LIN {X 0,Y 572.631,Z 334.16,A -85,B 0,C 180,E1 -2364.976,E2 -2364.976} C_VEL
LIN {X 0,Y 569.788,Z 334.515,A -85,B 0,C 180,E1 -2365.927,E2 -2365.927} C_VEL
LIN {X 0,Y 567.355,Z 334.817,A -85,B 0,C 180,E1 -2366.692,E2 -2366.692} C_VEL
LIN {X 0,Y 566.3,Z 334.946,A -85,B 0,C 180,E1 -2367.283,E2 -2367.283} C_VEL
LIN {X 0,Y 566.21,Z 334.956,A -85,B 0,C 180,E1 -2367.484,E2 -2367.484} C_VEL
LIN {X 0,Y 566.206,Z 334.958,A -85,B 0,C 180,E1 -2369.769,E2 -2369.769} C_VEL
LIN {X 0,Y 566.212,Z 334.959,A -85,B 0,C 180,E1 -2372.43,E2 -2372.43} C_VEL
LIN {X 0,Y 566.189,Z 334.96,A -85,B 0,C 180,E1 -2374.99,E2 -2374.99} C_VEL
LIN {X 0,Y 566.203,Z 334.958,A -85,B 0,C 180,E1 -2377.461,E2 -2377.461} C_VEL
LIN {X 0,Y 566.235,Z 334.956,A -85,B 0,C 180,E1 -2380.197,E2 -2380.197} C_VEL
LIN {X 0,Y 566.207,Z 334.957,A -85,B 0,C 180,E1 -2383.054,E2 -2383.054} C_VEL
LIN {X 0,Y 566.209,Z 334.958,A -85,B 0,C 180,E1 -2386.048,E2 -2386.048} C_VEL
LIN {X 0,Y 566.19,Z 334.959,A -85,B 0,C 180,E1 -2388.861,E2 -2388.861} C_VEL
LIN {X 0,Y 566.189,Z 334.961,A -85,B 0,C 180,E1 -2391.636,E2 -2391.636} C_VEL
LIN {X 0,Y 566.158,Z 334.963,A -85,B 0,C 180,E1 -2394.307,E2 -2394.307} C_VEL
LIN {X 0,Y 566.237,Z 334.955,A -85,B 0,C 180,E1 -2396.898,E2 -2396.898} C_VEL
LIN {X 0,Y 566.18,Z 334.963,A -85,B 0,C 180,E1 -2399.407,E2 -2399.407} C_VEL
LIN {X 0,Y 566.219,Z 334.956,A -85,B 0,C 180,E1 -2401.857,E2 -2401.857} C_VEL
LIN {X 0,Y 566.222,Z 334.955,A -85,B 0,C 180,E1 -2404.251,E2 -2404.251} C_VEL
LIN {X 0,Y 566.18,Z 334.961,A -85,B 0,C 180,E1 -2406.718,E2 -2406.718} C_VEL
LIN {X 0,Y 566.215,Z 334.957,A -85,B 0,C 180,E1 -2409.662,E2 -2409.662} C_VEL
LIN {X 0,Y 566.208,Z 334.959,A -85,B 0,C 180,E1 -2412.668,E2 -2412.668} C_VEL
LIN {X 0,Y 566.242,Z 334.952,A -85,B 0,C 180,E1 -2415.626,E2 -2415.626} C_VEL
LIN {X 0,Y 566.243,Z 334.954,A -85,B 0,C 180,E1 -2418.675,E2 -2418.675} C_VEL
LIN {X 0,Y 566.235,Z 334.954,A -85,B 0,C 180,E1 -2421.434,E2 -2421.434} C_VEL
LIN {X 0,Y 566.259,Z 334.952,A -85,B 0,C 180,E1 -2424.301,E2 -2424.301} C_VEL
LIN {X 0,Y 566.209,Z 334.958,A -85,B 0,C 180,E1 -2425.639,E2 -2425.639} C_VEL
LIN {X 0,Y 566.84,Z 337.939,A -85,B 0,C 180,E1 -2425.755,E2 -2425.755} C_VEL
LIN {X 0,Y 566.738,Z 351.089,A -85,B 0,C 180,E1 -2426.222,E2 -2426.222} C_VEL
LIN {X 0,Y 566.593,Z 362.987,A -85,B 0,C 180,E1 -2426.8,E2 -2426.8} C_VEL
LIN {X 0,Y 566.439,Z 374.351,A -85,B 0,C 180,E1 -2427.511,E2 -2427.511} C_VEL
LIN {X 0,Y 566.31,Z 384.605,A -85,B 0,C 180,E1 -2428.31,E2 -2428.31} C_VEL
LIN {X 0,Y 566.199,Z 393.028,A -85,B 0,C 180,E1 -2429.11,E2 -2429.11} C_VEL
LIN {X 0,Y 566.12,Z 400.82,A -85,B 0,C 180,E1 -2429.999,E2 -2429.999} C_VEL
LIN {X 0,Y 566.031,Z 408.464,A -85,B 0,C 180,E1 -2431.067,E2 -2431.067} C_VEL
LIN {X 0,Y 565.913,Z 414.624,A -85,B 0,C 180,E1 -2432.135,E2 -2432.135} C_VEL
LIN {X 0,Y 565.934,Z 419.527,A -85,B 0,C 180,E1 -2433.203,E2 -2433.203} C_VEL
LIN {X 0,Y 565.937,Z 423.326,A -85,B 0,C 180,E1 -2434.273,E2 -2434.273} C_VEL
LIN {X 0,Y 565.854,Z 425.292,A -85,B 0,C 180,E1 -2434.987,E2 -2434.987} C_VEL
LIN {X 0,Y 565.905,Z 426.839,A -85,B 0,C 180,E1 -2435.701,E2 -2435.701} C_VEL
LIN {X 0,Y 565.92,Z 428.087,A -85,B 0,C 180,E1 -2436.533,E2 -2436.533} C_VEL
LIN {X 0,Y 565.879,Z 428.964,A -85,B 0,C 180,E1 -2437.852,E2 -2437.852} C_VEL
LIN {X 0,Y 565.852,Z 428.889,A -85,B 0,C 180,E1 -2438.571,E2 -2438.571} C_VEL
LIN {X 0,Y 565.829,Z 428.38,A -85,B 0,C 180,E1 -2439.292,E2 -2439.292} C_VEL
LIN {X 0,Y 565.883,Z 427.462,A -85,B 0,C 180,E1 -2440.013,E2 -2440.013} C_VEL
LIN {X 0,Y 565.904,Z 425.165,A -85,B 0,C 180,E1 -2441.153,E2 -2441.153} C_VEL
LIN {X 0,Y 565.925,Z 422.132,A -85,B 0,C 180,E1 -2442.187,E2 -2442.187} C_VEL
LIN {X 0,Y 565.937,Z 417.853,A -85,B 0,C 180,E1 -2443.281,E2 -2443.281} C_VEL
LIN {X 0,Y 565.989,Z 412.171,A -85,B 0,C 180,E1 -2444.408,E2 -2444.408} C_VEL
LIN {X 0,Y 566.051,Z 405.374,A -85,B 0,C 180,E1 -2445.482,E2 -2445.482} C_VEL
LIN {X 0,Y 566.15,Z 398.227,A -85,B 0,C 180,E1 -2446.404,E2 -2446.404} C_VEL
LIN {X 0,Y 566.256,Z 389.547,A -85,B 0,C 180,E1 -2447.329,E2 -2447.329} C_VEL
LIN {X 0,Y 566.394,Z 378.723,A -85,B 0,C 180,E1 -2448.258,E2 -2448.258} C_VEL
LIN {X 0,Y 566.52,Z 368.124,A -85,B 0,C 180,E1 -2448.99,E2 -2448.99} C_VEL
LIN {X 0,Y 566.679,Z 357.756,A -85,B 0,C 180,E1 -2449.563,E2 -2449.563} C_VEL
LIN {X 0,Y 566.755,Z 345.733,A -85,B 0,C 180,E1 -2450.08,E2 -2450.08} C_VEL
LIN {X 0,Y 566.807,Z 337.369,A -85,B 0,C 180,E1 -2450.352,E2 -2450.352} C_VEL
LIN {X 0,Y 566.225,Z 334.958,A -85,B 0,C 180,E1 -2450.455,E2 -2450.455} C_VEL
LIN {X 0,Y 566.174,Z 334.963,A -85,B 0,C 180,E1 -2453.404,E2 -2453.404} C_VEL
LIN {X 0,Y 566.217,Z 334.958,A -85,B 0,C 180,E1 -2455.748,E2 -2455.748} C_VEL
LIN {X 0,Y 566.205,Z 334.959,A -85,B 0,C 180,E1 -2458.201,E2 -2458.201} C_VEL
LIN {X 0,Y 566.193,Z 334.959,A -85,B 0,C 180,E1 -2461.076,E2 -2461.076} C_VEL
LIN {X 0,Y 566.214,Z 334.958,A -85,B 0,C 180,E1 -2463.733,E2 -2463.733} C_VEL
LIN {X 0,Y 566.201,Z 334.961,A -85,B 0,C 180,E1 -2466.569,E2 -2466.569} C_VEL
LIN {X 0,Y 566.217,Z 334.957,A -85,B 0,C 180,E1 -2469.685,E2 -2469.685} C_VEL
LIN {X 0,Y 566.216,Z 334.956,A -85,B 0,C 180,E1 -2472.086,E2 -2472.086} C_VEL
LIN {X 0,Y 566.174,Z 334.962,A -85,B 0,C 180,E1 -2475.035,E2 -2475.035} C_VEL
LIN {X 0,Y 566.219,Z 334.957,A -85,B 0,C 180,E1 -2478.135,E2 -2478.135} C_VEL
LIN {X 0,Y 566.223,Z 334.956,A -85,B 0,C 180,E1 -2480.727,E2 -2480.727} C_VEL
LIN {X 0,Y 566.218,Z 334.956,A -85,B 0,C 180,E1 -2483.783,E2 -2483.783} C_VEL
LIN {X 0,Y 566.229,Z 334.956,A -85,B 0,C 180,E1 -2486.262,E2 -2486.262} C_VEL
LIN {X 0,Y 566.203,Z 334.955,A -85,B 0,C 180,E1 -2488.921,E2 -2488.921} C_VEL
LIN {X 0,Y 566.197,Z 334.955,A -85,B 0,C 180,E1 -2491.047,E2 -2491.047} C_VEL
LIN {X 0,Y 566.247,Z 334.954,A -85,B 0,C 180,E1 -2493.46,E2 -2493.46} C_VEL
LIN {X 0,Y 566.199,Z 334.958,A -85,B 0,C 180,E1 -2495.819,E2 -2495.819} C_VEL
LIN {X 0,Y 566.216,Z 334.956,A -85,B 0,C 180,E1 -2498.902,E2 -2498.902} C_VEL
LIN {X 0,Y 566.213,Z 334.957,A -85,B 0,C 180,E1 -2501.172,E2 -2501.172} C_VEL
LIN {X 0,Y 566.222,Z 334.958,A -85,B 0,C 180,E1 -2503.412,E2 -2503.412} C_VEL
LIN {X 0,Y 566.201,Z 334.961,A -85,B 0,C 180,E1 -2506.359,E2 -2506.359} C_VEL
LIN {X 0,Y 566.274,Z 334.95,A -85,B 0,C 180,E1 -2508.654,E2 -2508.654} C_VEL
LIN {X 0,Y 566.248,Z 334.954,A -85,B 0,C 180,E1 -2511.434,E2 -2511.434} C_VEL
LIN {X 0,Y 566.259,Z 334.952,A -85,B 0,C 180,E1 -2514.302,E2 -2514.302} C_VEL
LIN {X 0,Y 566.278,Z 334.949,A -85,B 0,C 180,E1 -2517.866,E2 -2517.866} C_VEL
LIN {X 0,Y 566.305,Z 334.945,A -85,B 0,C 180,E1 -2520.711,E2 -2520.711} C_VEL
LIN {X 0,Y 566.275,Z 334.949,A -85,B 0,C 180,E1 -2522.845,E2 -2522.845} C_VEL
LIN {X 0,Y 566.26,Z 334.95,A -85,B 0,C 180,E1 -2525.698,E2 -2525.698} C_VEL
LIN {X 0,Y 566.232,Z 334.955,A -85,B 0,C 180,E1 -2528.566,E2 -2528.566} C_VEL
LIN {X 0,Y 566.239,Z 334.955,A -85,B 0,C 180,E1 -2531.454,E2 -2531.454} C_VEL
LIN {X 0,Y 566.231,Z 334.955,A -85,B 0,C 180,E1 -2534.507,E2 -2534.507} C_VEL
LIN {X 0,Y 566.2,Z 334.959,A -85,B 0,C 180,E1 -2537.332,E2 -2537.332} C_VEL
LIN {X 0,Y 566.211,Z 334.958,A -85,B 0,C 180,E1 -2540.337,E2 -2540.337} C_VEL
LIN {X 0,Y 566.187,Z 334.961,A -85,B 0,C 180,E1 -2543.404,E2 -2543.404} C_VEL
LIN {X 0,Y 566.222,Z 334.956,A -85,B 0,C 180,E1 -2545.749,E2 -2545.749} C_VEL
LIN {X 0,Y 566.203,Z 334.961,A -85,B 0,C 180,E1 -2548.203,E2 -2548.203} C_VEL
LIN {X 0,Y 566.193,Z 334.96,A -85,B 0,C 180,E1 -2550.592,E2 -2550.592} C_VEL
LIN {X 0,Y 566.227,Z 334.958,A -85,B 0,C 180,E1 -2553.102,E2 -2553.102} C_VEL
LIN {X 0,Y 566.211,Z 334.957,A -85,B 0,C 180,E1 -2555.689,E2 -2555.689} C_VEL
LIN {X 0,Y 566.217,Z 334.955,A -85,B 0,C 180,E1 -2558.56,E2 -2558.56} C_VEL
LIN {X 0,Y 566.22,Z 334.957,A -85,B 0,C 180,E1 -2561.136,E2 -2561.136} C_VEL
LIN {X 0,Y 566.199,Z 334.96,A -85,B 0,C 180,E1 -2564.036,E2 -2564.036} C_VEL
LIN {X 0,Y 566.214,Z 334.958,A -85,B 0,C 180,E1 -2567.082,E2 -2567.082} C_VEL
LIN {X 0,Y 566.227,Z 334.957,A -85,B 0,C 180,E1 -2569.803,E2 -2569.803} C_VEL
LIN {X 0,Y 566.199,Z 334.96,A -85,B 0,C 180,E1 -2572.599,E2 -2572.599} C_VEL
LIN {X 0,Y 566.293,Z 335.146,A -85,B 0,C 180,E1 -2573.272,E2 -2573.272} C_VEL
LIN {X 0,Y 567.038,Z 340.964,A -85,B 0,C 180,E1 -2574.672,E2 -2574.672} C_VEL
LIN {X 0,Y 566.802,Z 353.562,A -85,B 0,C 180,E1 -2577.475,E2 -2577.475} C_VEL
LIN {X 0,Y 566.768,Z 366.586,A -85,B 0,C 180,E1 -2580.265,E2 -2580.265} C_VEL
LIN {X 0,Y 566.756,Z 379.73,A -85,B 0,C 180,E1 -2583.001,E2 -2583.001} C_VEL
LIN {X 0,Y 566.697,Z 393.877,A -85,B 0,C 180,E1 -2585.842,E2 -2585.842} C_VEL
LIN {X 0,Y 566.601,Z 405.015,A -85,B 0,C 180,E1 -2588.155,E2 -2588.155} C_VEL
LIN {X 0,Y 566.386,Z 419.542,A -85,B 0,C 180,E1 -2591.179,E2 -2591.179} C_VEL
LIN {X 0,Y 566.26,Z 432.253,A -85,B 0,C 180,E1 -2593.785,E2 -2593.785} C_VEL
LIN {X 0,Y 566.18,Z 444.964,A -85,B 0,C 180,E1 -2596.359,E2 -2596.359} C_VEL
LIN {X 0,Y 566.158,Z 449.882,A -85,B 0,C 180,E1 -2597.306,E2 -2597.306} C_VEL
LIN {X 0,Y 566.95,Z 456.115,A -85,B 0,C 180,E1 -2597.426,E2 -2597.426} C_VEL
LIN {X 0,Y 566.851,Z 468.998,A -85,B 0,C 180,E1 -2597.742,E2 -2597.742} C_VEL
LIN {X 0,Y 566.724,Z 481.507,A -85,B 0,C 180,E1 -2598.194,E2 -2598.194} C_VEL
LIN {X 0,Y 566.618,Z 493.248,A -85,B 0,C 180,E1 -2598.77,E2 -2598.77} C_VEL
LIN {X 0,Y 566.454,Z 504.208,A -85,B 0,C 180,E1 -2599.456,E2 -2599.456} C_VEL
LIN {X 0,Y 566.327,Z 514.607,A -85,B 0,C 180,E1 -2600.266,E2 -2600.266} C_VEL
LIN {X 0,Y 566.207,Z 523.118,A -85,B 0,C 180,E1 -2601.075,E2 -2601.075} C_VEL
LIN {X 0,Y 566.112,Z 530.965,A -85,B 0,C 180,E1 -2601.972,E2 -2601.972} C_VEL
LIN {X 0,Y 566,Z 538.625,A -85,B 0,C 180,E1 -2603.047,E2 -2603.047} C_VEL
LIN {X 0,Y 566.004,Z 545.683,A -85,B 0,C 180,E1 -2604.3,E2 -2604.3} C_VEL
LIN {X 0,Y 565.933,Z 550.374,A -85,B 0,C 180,E1 -2605.371,E2 -2605.371} C_VEL
LIN {X 0,Y 565.926,Z 553.959,A -85,B 0,C 180,E1 -2606.441,E2 -2606.441} C_VEL
LIN {X 0,Y 565.878,Z 555.809,A -85,B 0,C 180,E1 -2607.153,E2 -2607.153} C_VEL
LIN {X 0,Y 565.846,Z 558.186,A -85,B 0,C 180,E1 -2608.577,E2 -2608.577} C_VEL
LIN {X 0,Y 565.839,Z 559,A -85,B 0,C 180,E1 -2610.001,E2 -2610.001} C_VEL
LIN {X 0,Y 565.846,Z 558.186,A -85,B 0,C 180,E1 -2611.424,E2 -2611.424} C_VEL
LIN {X 0,Y 565.878,Z 555.809,A -85,B 0,C 180,E1 -2612.848,E2 -2612.848} C_VEL
LIN {X 0,Y 565.926,Z 552.894,A -85,B 0,C 180,E1 -2613.917,E2 -2613.917} C_VEL
LIN {X 0,Y 565.878,Z 548.947,A -85,B 0,C 180,E1 -2614.988,E2 -2614.988} C_VEL
LIN {X 0,Y 566.002,Z 543.864,A -85,B 0,C 180,E1 -2616.059,E2 -2616.059} C_VEL
LIN {X 0,Y 566.041,Z 537.465,A -85,B 0,C 180,E1 -2617.133,E2 -2617.133} C_VEL
LIN {X 0,Y 566.134,Z 529.474,A -85,B 0,C 180,E1 -2618.208,E2 -2618.208} C_VEL
LIN {X 0,Y 566.229,Z 521.33,A -85,B 0,C 180,E1 -2619.106,E2 -2619.106} C_VEL
LIN {X 0,Y 566.35,Z 511.394,A -85,B 0,C 180,E1 -2620.005,E2 -2620.005} C_VEL
LIN {X 0,Y 566.523,Z 500.282,A -85,B 0,C 180,E1 -2620.808,E2 -2620.808} C_VEL
LIN {X 0,Y 566.613,Z 489.167,A -85,B 0,C 180,E1 -2621.447,E2 -2621.447} C_VEL
LIN {X 0,Y 566.741,Z 476.971,A -85,B 0,C 180,E1 -2621.989,E2 -2621.989} C_VEL
LIN {X 0,Y 566.879,Z 464.155,A -85,B 0,C 180,E1 -2622.395,E2 -2622.395} C_VEL
LIN {X 0,Y 566.758,Z 453.575,A -85,B 0,C 180,E1 -2622.625,E2 -2622.625} C_VEL
LIN {X 0,Y 566.146,Z 449.612,A -85,B 0,C 180,E1 -2622.707,E2 -2622.707} C_VEL
LIN {X 0,Y 566.251,Z 435.879,A -85,B 0,C 180,E1 -2625.477,E2 -2625.477} C_VEL
LIN {X 0,Y 566.366,Z 423.168,A -85,B 0,C 180,E1 -2628.073,E2 -2628.073} C_VEL
LIN {X 0,Y 566.489,Z 410.457,A -85,B 0,C 180,E1 -2630.707,E2 -2630.707} C_VEL
LIN {X 0,Y 566.689,Z 397.641,A -85,B 0,C 180,E1 -2633.402,E2 -2633.402} C_VEL
LIN {X 0,Y 566.752,Z 382.192,A -85,B 0,C 180,E1 -2636.515,E2 -2636.515} C_VEL
LIN {X 0,Y 566.78,Z 368.63,A -85,B 0,C 180,E1 -2639.328,E2 -2639.328} C_VEL
LIN {X 0,Y 566.833,Z 355.117,A -85,B 0,C 180,E1 -2642.219,E2 -2642.219} C_VEL
LIN {X 0,Y 567.083,Z 342.053,A -85,B 0,C 180,E1 -2645.119,E2 -2645.119} C_VEL
LIN {X 0,Y 566.832,Z 338.493,A -85,B 0,C 180,E1 -2645.948,E2 -2645.948} C_VEL
LIN {X 0,Y 566.222,Z 334.958,A -85,B 0,C 180,E1 -2646.846,E2 -2646.846} C_VEL
LIN {X 0,Y 566.218,Z 334.957,A -85,B 0,C 180,E1 -2649.686,E2 -2649.686} C_VEL
LIN {X 0,Y 566.22,Z 334.956,A -85,B 0,C 180,E1 -2652.087,E2 -2652.087} C_VEL
LIN {X 0,Y 566.179,Z 334.964,A -85,B 0,C 180,E1 -2655.036,E2 -2655.036} C_VEL
LIN {X 0,Y 566.193,Z 334.958,A -85,B 0,C 180,E1 -2657.911,E2 -2657.911} C_VEL
LIN {X 0,Y 566.228,Z 334.957,A -85,B 0,C 180,E1 -2660.727,E2 -2660.727} C_VEL
LIN {X 0,Y 566.189,Z 334.961,A -85,B 0,C 180,E1 -2663.788,E2 -2663.788} C_VEL
LIN {X 0,Y 566.217,Z 334.958,A -85,B 0,C 180,E1 -2666.266,E2 -2666.266} C_VEL
LIN {X 0,Y 566.205,Z 334.958,A -85,B 0,C 180,E1 -2668.922,E2 -2668.922} C_VEL
LIN {X 0,Y 566.217,Z 334.958,A -85,B 0,C 180,E1 -2671.858,E2 -2671.858} C_VEL
LIN {X 0,Y 566.215,Z 334.958,A -85,B 0,C 180,E1 -2674.251,E2 -2674.251} C_VEL
LIN {X 0,Y 566.198,Z 334.959,A -85,B 0,C 180,E1 -2676.714,E2 -2676.714} C_VEL
LIN {X 0,Y 566.212,Z 334.959,A -85,B 0,C 180,E1 -2679.663,E2 -2679.663} C_VEL
LIN {X 0,Y 566.204,Z 334.958,A -85,B 0,C 180,E1 -2682.669,E2 -2682.669} C_VEL
LIN {X 0,Y 566.24,Z 334.953,A -85,B 0,C 180,E1 -2685.627,E2 -2685.627} C_VEL
LIN {X 0,Y 566.241,Z 334.956,A -85,B 0,C 180,E1 -2688.676,E2 -2688.676} C_VEL
LIN {X 0,Y 566.234,Z 334.953,A -85,B 0,C 180,E1 -2691.435,E2 -2691.435} C_VEL
LIN {X 0,Y 566.264,Z 334.953,A -85,B 0,C 180,E1 -2694.302,E2 -2694.302} C_VEL
LIN {X 0,Y 566.28,Z 334.95,A -85,B 0,C 180,E1 -2697.866,E2 -2697.866} C_VEL
LIN {X 0,Y 566.31,Z 334.945,A -85,B 0,C 180,E1 -2700.711,E2 -2700.711} C_VEL
LIN {X 0,Y 566.278,Z 334.948,A -85,B 0,C 180,E1 -2702.846,E2 -2702.846} C_VEL
LIN {X 0,Y 566.261,Z 334.952,A -85,B 0,C 180,E1 -2705.698,E2 -2705.698} C_VEL
LIN {X 0,Y 566.24,Z 334.954,A -85,B 0,C 180,E1 -2708.566,E2 -2708.566} C_VEL
LIN {X 0,Y 566.249,Z 334.953,A -85,B 0,C 180,E1 -2711.454,E2 -2711.454} C_VEL
LIN {X 0,Y 566.241,Z 334.955,A -85,B 0,C 180,E1 -2714.507,E2 -2714.507} C_VEL
LIN {X 0,Y 566.21,Z 334.957,A -85,B 0,C 180,E1 -2717.332,E2 -2717.332} C_VEL
LIN {X 0,Y 566.213,Z 334.957,A -85,B 0,C 180,E1 -2720.337,E2 -2720.337} C_VEL
LIN {X 0,Y 566.196,Z 334.961,A -85,B 0,C 180,E1 -2723.404,E2 -2723.404} C_VEL
LIN {X 0,Y 566.222,Z 334.958,A -85,B 0,C 180,E1 -2725.749,E2 -2725.749} C_VEL
LIN {X 0,Y 566.21,Z 334.956,A -85,B 0,C 180,E1 -2727.484,E2 -2727.484} C_VEL
LIN {X 0,Y 565.529,Z 335.043,A -85,B 0,C 180,E1 -2728.077,E2 -2728.077} C_VEL
LIN {X 0,Y 562.663,Z 335.401,A -85,B 0,C 180,E1 -2729.041,E2 -2729.041} C_VEL
LIN {X 0,Y 560.253,Z 335.7,A -85,B 0,C 180,E1 -2729.817,E2 -2729.817} C_VEL
LIN {X 0,Y 559.226,Z 335.827,A -85,B 0,C 180,E1 -2730.415,E2 -2730.415} C_VEL
LIN {X 0,Y 559.146,Z 335.836,A -85,B 0,C 180,E1 -2730.618,E2 -2730.618} C_VEL
LIN {X 0,Y 559.172,Z 335.836,A -85,B 0,C 180,E1 -2733.575,E2 -2733.575} C_VEL
LIN {X 0,Y 559.153,Z 335.835,A -85,B 0,C 180,E1 -2736.445,E2 -2736.445} C_VEL
LIN {X 0,Y 559.186,Z 335.832,A -85,B 0,C 180,E1 -2738.934,E2 -2738.934} C_VEL
LIN {X 0,Y 559.173,Z 335.834,A -85,B 0,C 180,E1 -2741.77,E2 -2741.77} C_VEL
LIN {X 0,Y 559.142,Z 335.839,A -85,B 0,C 180,E1 -2744.74,E2 -2744.74} C_VEL
LIN {X 0,Y 559.185,Z 335.833,A -85,B 0,C 180,E1 -2747.862,E2 -2747.862} C_VEL
LIN {X 0,Y 559.179,Z 335.833,A -85,B 0,C 180,E1 -2751.066,E2 -2751.066} C_VEL
LIN {X 0,Y 559.128,Z 335.841,A -85,B 0,C 180,E1 -2753.788,E2 -2753.788} C_VEL
LIN {X 0,Y 559.172,Z 335.833,A -85,B 0,C 180,E1 -2756.425,E2 -2756.425} C_VEL
LIN {X 0,Y 559.158,Z 335.836,A -85,B 0,C 180,E1 -2758.98,E2 -2758.98} C_VEL
LIN {X 0,Y 559.175,Z 335.835,A -85,B 0,C 180,E1 -2761.619,E2 -2761.619} C_VEL
LIN {X 0,Y 559.189,Z 335.833,A -85,B 0,C 180,E1 -2763.903,E2 -2763.903} C_VEL
LIN {X 0,Y 559.15,Z 335.836,A -85,B 0,C 180,E1 -2766.571,E2 -2766.571} C_VEL
LIN {X 0,Y 559.184,Z 335.835,A -85,B 0,C 180,E1 -2769.395,E2 -2769.395} C_VEL
LIN {X 0,Y 559.151,Z 335.838,A -85,B 0,C 180,E1 -2771.685,E2 -2771.685} C_VEL
LIN {X 0,Y 559.173,Z 335.835,A -85,B 0,C 180,E1 -2773.948,E2 -2773.948} C_VEL
LIN {X 0,Y 559.178,Z 335.835,A -85,B 0,C 180,E1 -2776.184,E2 -2776.184} C_VEL
LIN {X 0,Y 559.204,Z 335.83,A -85,B 0,C 180,E1 -2779.133,E2 -2779.133} C_VEL
LIN {X 0,Y 559.212,Z 335.829,A -85,B 0,C 180,E1 -2782.053,E2 -2782.053} C_VEL
LIN {X 0,Y 559.255,Z 335.825,A -85,B 0,C 180,E1 -2784.953,E2 -2784.953} C_VEL
LIN {X 0,Y 559.16,Z 335.837,A -85,B 0,C 180,E1 -2785.517,E2 -2785.517} C_VEL
LIN {X 0,Y 559.881,Z 339.83,A -85,B 0,C 180,E1 -2785.658,E2 -2785.658} C_VEL
LIN {X 0,Y 559.768,Z 352.4,A -85,B 0,C 180,E1 -2786.13,E2 -2786.13} C_VEL
LIN {X 0,Y 559.596,Z 364.752,A -85,B 0,C 180,E1 -2786.76,E2 -2786.76} C_VEL
LIN {X 0,Y 559.424,Z 375.787,A -85,B 0,C 180,E1 -2787.479,E2 -2787.479} C_VEL
LIN {X 0,Y 559.298,Z 384.746,A -85,B 0,C 180,E1 -2788.199,E2 -2788.199} C_VEL
LIN {X 0,Y 559.137,Z 393.997,A -85,B 0,C 180,E1 -2789.099,E2 -2789.099} C_VEL
LIN {X 0,Y 559.033,Z 402.956,A -85,B 0,C 180,E1 -2790.18,E2 -2790.18} C_VEL
LIN {X 0,Y 558.926,Z 410.206,A -85,B 0,C 180,E1 -2791.26,E2 -2791.26} C_VEL
LIN {X 0,Y 558.855,Z 416.871,A -85,B 0,C 180,E1 -2792.522,E2 -2792.522} C_VEL
LIN {X 0,Y 558.858,Z 421.288,A -85,B 0,C 180,E1 -2793.605,E2 -2793.605} C_VEL
LIN {X 0,Y 558.828,Z 423.628,A -85,B 0,C 180,E1 -2794.327,E2 -2794.327} C_VEL
LIN {X 0,Y 558.769,Z 425.543,A -85,B 0,C 180,E1 -2795.051,E2 -2795.051} C_VEL
LIN {X 0,Y 558.816,Z 427.028,A -85,B 0,C 180,E1 -2795.774,E2 -2795.774} C_VEL
LIN {X 0,Y 558.848,Z 428.109,A -85,B 0,C 180,E1 -2796.535,E2 -2796.535} C_VEL
LIN {X 0,Y 558.797,Z 428.986,A -85,B 0,C 180,E1 -2797.952,E2 -2797.952} C_VEL
LIN {X 0,Y 558.766,Z 428.841,A -85,B 0,C 180,E1 -2798.68,E2 -2798.68} C_VEL
LIN {X 0,Y 558.78,Z 427.299,A -85,B 0,C 180,E1 -2800.141,E2 -2800.141} C_VEL
LIN {X 0,Y 558.806,Z 425.178,A -85,B 0,C 180,E1 -2801.187,E2 -2801.187} C_VEL
LIN {X 0,Y 558.835,Z 421.774,A -85,B 0,C 180,E1 -2802.344,E2 -2802.344} C_VEL
LIN {X 0,Y 558.851,Z 417.385,A -85,B 0,C 180,E1 -2803.453,E2 -2803.453} C_VEL
LIN {X 0,Y 558.919,Z 411.747,A -85,B 0,C 180,E1 -2804.565,E2 -2804.565} C_VEL
LIN {X 0,Y 558.989,Z 404.648,A -85,B 0,C 180,E1 -2805.682,E2 -2805.682} C_VEL
LIN {X 0,Y 559.117,Z 395.668,A -85,B 0,C 180,E1 -2806.804,E2 -2806.804} C_VEL
LIN {X 0,Y 559.3,Z 386.408,A -85,B 0,C 180,E1 -2807.741,E2 -2807.741} C_VEL
LIN {X 0,Y 559.428,Z 376.091,A -85,B 0,C 180,E1 -2808.589,E2 -2808.589} C_VEL
LIN {X 0,Y 559.631,Z 364.33,A -85,B 0,C 180,E1 -2809.354,E2 -2809.354} C_VEL
LIN {X 0,Y 559.783,Z 352.449,A -85,B 0,C 180,E1 -2809.958,E2 -2809.958} C_VEL
LIN {X 0,Y 559.877,Z 339.819,A -85,B 0,C 180,E1 -2810.433,E2 -2810.433} C_VEL
LIN {X 0,Y 559.196,Z 335.891,A -85,B 0,C 180,E1 -2810.567,E2 -2810.567} C_VEL
LIN {X 0,Y 559.141,Z 335.839,A -85,B 0,C 180,E1 -2813.716,E2 -2813.716} C_VEL
LIN {X 0,Y 559.182,Z 335.833,A -85,B 0,C 180,E1 -2816.096,E2 -2816.096} C_VEL
LIN {X 0,Y 559.166,Z 335.837,A -85,B 0,C 180,E1 -2818.529,E2 -2818.529} C_VEL
LIN {X 0,Y 559.148,Z 335.837,A -85,B 0,C 180,E1 -2821.273,E2 -2821.273} C_VEL
LIN {X 0,Y 559.168,Z 335.834,A -85,B 0,C 180,E1 -2823.949,E2 -2823.949} C_VEL
LIN {X 0,Y 559.142,Z 335.838,A -85,B 0,C 180,E1 -2827.108,E2 -2827.108} C_VEL
LIN {X 0,Y 559.162,Z 335.835,A -85,B 0,C 180,E1 -2829.941,E2 -2829.941} C_VEL
LIN {X 0,Y 559.165,Z 335.836,A -85,B 0,C 180,E1 -2832.742,E2 -2832.742} C_VEL
LIN {X 0,Y 559.153,Z 335.837,A -85,B 0,C 180,E1 -2835.76,E2 -2835.76} C_VEL
LIN {X 0,Y 559.192,Z 335.833,A -85,B 0,C 180,E1 -2838.232,E2 -2838.232} C_VEL
LIN {X 0,Y 559.179,Z 335.834,A -85,B 0,C 180,E1 -2841.19,E2 -2841.19} C_VEL
LIN {X 0,Y 559.173,Z 335.833,A -85,B 0,C 180,E1 -2843.791,E2 -2843.791} C_VEL
LIN {X 0,Y 559.178,Z 335.835,A -85,B 0,C 180,E1 -2846.426,E2 -2846.426} C_VEL
LIN {X 0,Y 559.167,Z 335.831,A -85,B 0,C 180,E1 -2848.981,E2 -2848.981} C_VEL
LIN {X 0,Y 559.171,Z 335.833,A -85,B 0,C 180,E1 -2851.617,E2 -2851.617} C_VEL
LIN {X 0,Y 559.2,Z 335.83,A -85,B 0,C 180,E1 -2853.904,E2 -2853.904} C_VEL
LIN {X 0,Y 559.156,Z 335.835,A -85,B 0,C 180,E1 -2856.567,E2 -2856.567} C_VEL
LIN {X 0,Y 559.186,Z 335.835,A -85,B 0,C 180,E1 -2859.395,E2 -2859.395} C_VEL
LIN {X 0,Y 559.155,Z 335.835,A -85,B 0,C 180,E1 -2861.686,E2 -2861.686} C_VEL
LIN {X 0,Y 559.172,Z 335.834,A -85,B 0,C 180,E1 -2863.948,E2 -2863.948} C_VEL
LIN {X 0,Y 559.174,Z 335.835,A -85,B 0,C 180,E1 -2866.184,E2 -2866.184} C_VEL
LIN {X 0,Y 559.209,Z 335.83,A -85,B 0,C 180,E1 -2869.134,E2 -2869.134} C_VEL
LIN {X 0,Y 559.208,Z 335.83,A -85,B 0,C 180,E1 -2872.053,E2 -2872.053} C_VEL
LIN {X 0,Y 559.257,Z 335.822,A -85,B 0,C 180,E1 -2874.953,E2 -2874.953} C_VEL
LIN {X 0,Y 559.249,Z 335.824,A -85,B 0,C 180,E1 -2877.839,E2 -2877.839} C_VEL
LIN {X 0,Y 559.275,Z 335.82,A -85,B 0,C 180,E1 -2880.72,E2 -2880.72} C_VEL
LIN {X 0,Y 559.241,Z 335.826,A -85,B 0,C 180,E1 -2882.881,E2 -2882.881} C_VEL
LIN {X 0,Y 559.229,Z 335.826,A -85,B 0,C 180,E1 -2885.77,E2 -2885.77} C_VEL
LIN {X 0,Y 559.19,Z 335.831,A -85,B 0,C 180,E1 -2888.674,E2 -2888.674} C_VEL
LIN {X 0,Y 559.202,Z 335.83,A -85,B 0,C 180,E1 -2891.6,E2 -2891.6} C_VEL
LIN {X 0,Y 559.196,Z 335.831,A -85,B 0,C 180,E1 -2894.596,E2 -2894.596} C_VEL
LIN {X 0,Y 559.16,Z 335.835,A -85,B 0,C 180,E1 -2897.557,E2 -2897.557} C_VEL
LIN {X 0,Y 559.169,Z 335.835,A -85,B 0,C 180,E1 -2899.837,E2 -2899.837} C_VEL
LIN {X 0,Y 559.139,Z 335.84,A -85,B 0,C 180,E1 -2902.153,E2 -2902.153} C_VEL
LIN {X 0,Y 559.177,Z 335.836,A -85,B 0,C 180,E1 -2905.187,E2 -2905.187} C_VEL
LIN {X 0,Y 559.193,Z 335.832,A -85,B 0,C 180,E1 -2907.712,E2 -2907.712} C_VEL
LIN {X 0,Y 559.167,Z 335.838,A -85,B 0,C 180,E1 -2910.182,E2 -2910.182} C_VEL
LIN {X 0,Y 559.173,Z 335.834,A -85,B 0,C 180,E1 -2912.714,E2 -2912.714} C_VEL
LIN {X 0,Y 559.156,Z 335.837,A -85,B 0,C 180,E1 -2915.322,E2 -2915.322} C_VEL
LIN {X 0,Y 559.135,Z 335.84,A -85,B 0,C 180,E1 -2918.017,E2 -2918.017} C_VEL
LIN {X 0,Y 559.179,Z 335.834,A -85,B 0,C 180,E1 -2920.811,E2 -2920.811} C_VEL
LIN {X 0,Y 559.161,Z 335.835,A -85,B 0,C 180,E1 -2923.732,E2 -2923.732} C_VEL
LIN {X 0,Y 559.173,Z 335.833,A -85,B 0,C 180,E1 -2926.801,E2 -2926.801} C_VEL
LIN {X 0,Y 559.18,Z 335.836,A -85,B 0,C 180,E1 -2929.19,E2 -2929.19} C_VEL
LIN {X 0,Y 559.136,Z 335.842,A -85,B 0,C 180,E1 -2931.983,E2 -2931.983} C_VEL
LIN {X 0,Y 559.226,Z 335.98,A -85,B 0,C 180,E1 -2933.035,E2 -2933.035} C_VEL
LIN {X 0,Y 560.088,Z 341.038,A -85,B 0,C 180,E1 -2934.297,E2 -2934.297} C_VEL
LIN {X 0,Y 559.91,Z 350.543,A -85,B 0,C 180,E1 -2936.476,E2 -2936.476} C_VEL
LIN {X 0,Y 559.83,Z 364.036,A -85,B 0,C 180,E1 -2939.441,E2 -2939.441} C_VEL
LIN {X 0,Y 559.739,Z 377.565,A -85,B 0,C 180,E1 -2942.318,E2 -2942.318} C_VEL
LIN {X 0,Y 559.648,Z 391.261,A -85,B 0,C 180,E1 -2945.123,E2 -2945.123} C_VEL
LIN {X 0,Y 559.601,Z 404.875,A -85,B 0,C 180,E1 -2947.867,E2 -2947.867} C_VEL
LIN {X 0,Y 559.403,Z 419.542,A -85,B 0,C 180,E1 -2950.935,E2 -2950.935} C_VEL
LIN {X 0,Y 559.264,Z 432.253,A -85,B 0,C 180,E1 -2953.576,E2 -2953.576} C_VEL
LIN {X 0,Y 559.119,Z 446.78,A -85,B 0,C 180,E1 -2956.554,E2 -2956.554} C_VEL
LIN {X 0,Y 559.099,Z 449.882,A -85,B 0,C 180,E1 -2957.143,E2 -2957.143} C_VEL
LIN {X 0,Y 560.046,Z 457.255,A -85,B 0,C 180,E1 -2957.292,E2 -2957.292} C_VEL
LIN {X 0,Y 559.916,Z 470.518,A -85,B 0,C 180,E1 -2957.634,E2 -2957.634} C_VEL
LIN {X 0,Y 559.768,Z 482.533,A -85,B 0,C 180,E1 -2958.091,E2 -2958.091} C_VEL
LIN {X 0,Y 559.605,Z 495.277,A -85,B 0,C 180,E1 -2958.745,E2 -2958.745} C_VEL
LIN {X 0,Y 559.427,Z 506.753,A -85,B 0,C 180,E1 -2959.505,E2 -2959.505} C_VEL
LIN {X 0,Y 559.244,Z 517.606,A -85,B 0,C 180,E1 -2960.415,E2 -2960.415} C_VEL
LIN {X 0,Y 559.127,Z 526.418,A -85,B 0,C 180,E1 -2961.325,E2 -2961.325} C_VEL
LIN {X 0,Y 558.996,Z 535.005,A -85,B 0,C 180,E1 -2962.415,E2 -2962.415} C_VEL
LIN {X 0,Y 558.884,Z 542.69,A -85,B 0,C 180,E1 -2963.649,E2 -2963.649} C_VEL
LIN {X 0,Y 558.869,Z 547.368,A -85,B 0,C 180,E1 -2964.589,E2 -2964.589} C_VEL
LIN {X 0,Y 558.868,Z 551.679,A -85,B 0,C 180,E1 -2965.673,E2 -2965.673} C_VEL
LIN {X 0,Y 558.836,Z 553.959,A -85,B 0,C 180,E1 -2966.395,E2 -2966.395} C_VEL
LIN {X 0,Y 558.799,Z 555.809,A -85,B 0,C 180,E1 -2967.117,E2 -2967.117} C_VEL
LIN {X 0,Y 558.746,Z 558.186,A -85,B 0,C 180,E1 -2968.559,E2 -2968.559} C_VEL
LIN {X 0,Y 558.74,Z 559,A -85,B 0,C 180,E1 -2970.001,E2 -2970.001} C_VEL
LIN {X 0,Y 558.746,Z 558.185,A -85,B 0,C 180,E1 -2971.442,E2 -2971.442} C_VEL
LIN {X 0,Y 558.799,Z 555.809,A -85,B 0,C 180,E1 -2972.884,E2 -2972.884} C_VEL
LIN {X 0,Y 558.844,Z 552.894,A -85,B 0,C 180,E1 -2973.967,E2 -2973.967} C_VEL
LIN {X 0,Y 558.798,Z 548.947,A -85,B 0,C 180,E1 -2975.051,E2 -2975.051} C_VEL
LIN {X 0,Y 558.921,Z 543.864,A -85,B 0,C 180,E1 -2976.136,E2 -2976.136} C_VEL
LIN {X 0,Y 558.978,Z 537.464,A -85,B 0,C 180,E1 -2977.223,E2 -2977.223} C_VEL
LIN {X 0,Y 559.099,Z 529.474,A -85,B 0,C 180,E1 -2978.312,E2 -2978.312} C_VEL
LIN {X 0,Y 559.195,Z 521.33,A -85,B 0,C 180,E1 -2979.222,E2 -2979.222} C_VEL
LIN {X 0,Y 559.359,Z 511.394,A -85,B 0,C 180,E1 -2980.132,E2 -2980.132} C_VEL
LIN {X 0,Y 559.527,Z 500.39,A -85,B 0,C 180,E1 -2980.938,E2 -2980.938} C_VEL
LIN {X 0,Y 559.672,Z 488.451,A -85,B 0,C 180,E1 -2981.628,E2 -2981.628} C_VEL
LIN {X 0,Y 559.833,Z 475.753,A -85,B 0,C 180,E1 -2982.185,E2 -2982.185} C_VEL
LIN {X 0,Y 559.979,Z 462.326,A -85,B 0,C 180,E1 -2982.596,E2 -2982.596} C_VEL
LIN {X 0,Y 559.824,Z 454.3,A -85,B 0,C 180,E1 -2982.772,E2 -2982.772} C_VEL
LIN {X 0,Y 559.087,Z 449.612,A -85,B 0,C 180,E1 -2982.87,E2 -2982.87} C_VEL
LIN {X 0,Y 559.203,Z 435.879,A -85,B 0,C 180,E1 -2985.677,E2 -2985.677} C_VEL
LIN {X 0,Y 559.348,Z 423.168,A -85,B 0,C 180,E1 -2988.308,E2 -2988.308} C_VEL
LIN {X 0,Y 559.5,Z 410.457,A -85,B 0,C 180,E1 -2990.978,E2 -2990.978} C_VEL
LIN {X 0,Y 559.632,Z 399.415,A -85,B 0,C 180,E1 -2993.228,E2 -2993.228} C_VEL
LIN {X 0,Y 559.708,Z 385.472,A -85,B 0,C 180,E1 -2996.071,E2 -2996.071} C_VEL
LIN {X 0,Y 559.747,Z 371.89,A -85,B 0,C 180,E1 -2998.908,E2 -2998.908} C_VEL
LIN {X 0,Y 559.846,Z 360.352,A -85,B 0,C 180,E1 -3001.39,E2 -3001.39} C_VEL
LIN {X 0,Y 560.034,Z 346.932,A -85,B 0,C 180,E1 -3004.383,E2 -3004.383} C_VEL
LIN {X 0,Y 560.08,Z 341.151,A -85,B 0,C 180,E1 -3005.708,E2 -3005.708} C_VEL
LIN {X 0,Y 559.192,Z 335.834,A -85,B 0,C 180,E1 -3007.021,E2 -3007.021} C_VEL
LIN {X 0,Y 559.164,Z 335.835,A -85,B 0,C 180,E1 -3009.942,E2 -3009.942} C_VEL
LIN {X 0,Y 559.17,Z 335.837,A -85,B 0,C 180,E1 -3012.743,E2 -3012.743} C_VEL
LIN {X 0,Y 559.158,Z 335.835,A -85,B 0,C 180,E1 -3015.761,E2 -3015.761} C_VEL
LIN {X 0,Y 559.17,Z 335.835,A -85,B 0,C 180,E1 -3018.23,E2 -3018.23} C_VEL
LIN {X 0,Y 559.184,Z 335.832,A -85,B 0,C 180,E1 -3021.191,E2 -3021.191} C_VEL
LIN {X 0,Y 559.144,Z 335.838,A -85,B 0,C 180,E1 -3023.79,E2 -3023.79} C_VEL
LIN {X 0,Y 559.168,Z 335.836,A -85,B 0,C 180,E1 -3026.425,E2 -3026.425} C_VEL
LIN {X 0,Y 559.169,Z 335.834,A -85,B 0,C 180,E1 -3028.981,E2 -3028.981} C_VEL
LIN {X 0,Y 559.173,Z 335.834,A -85,B 0,C 180,E1 -3031.619,E2 -3031.619} C_VEL
LIN {X 0,Y 559.184,Z 335.833,A -85,B 0,C 180,E1 -3033.903,E2 -3033.903} C_VEL
LIN {X 0,Y 559.163,Z 335.836,A -85,B 0,C 180,E1 -3036.568,E2 -3036.568} C_VEL
LIN {X 0,Y 559.181,Z 335.833,A -85,B 0,C 180,E1 -3039.396,E2 -3039.396} C_VEL
LIN {X 0,Y 559.144,Z 335.837,A -85,B 0,C 180,E1 -3041.686,E2 -3041.686} C_VEL
LIN {X 0,Y 559.174,Z 335.834,A -85,B 0,C 180,E1 -3043.948,E2 -3043.948} C_VEL
LIN {X 0,Y 559.178,Z 335.833,A -85,B 0,C 180,E1 -3046.184,E2 -3046.184} C_VEL
LIN {X 0,Y 559.199,Z 335.83,A -85,B 0,C 180,E1 -3049.134,E2 -3049.134} C_VEL
LIN {X 0,Y 559.211,Z 335.831,A -85,B 0,C 180,E1 -3052.054,E2 -3052.054} C_VEL
LIN {X 0,Y 559.261,Z 335.822,A -85,B 0,C 180,E1 -3054.954,E2 -3054.954} C_VEL
LIN {X 0,Y 559.252,Z 335.825,A -85,B 0,C 180,E1 -3057.84,E2 -3057.84} C_VEL
LIN {X 0,Y 559.28,Z 335.821,A -85,B 0,C 180,E1 -3060.72,E2 -3060.72} C_VEL
LIN {X 0,Y 559.245,Z 335.825,A -85,B 0,C 180,E1 -3062.882,E2 -3062.882} C_VEL
LIN {X 0,Y 559.231,Z 335.827,A -85,B 0,C 180,E1 -3065.77,E2 -3065.77} C_VEL
LIN {X 0,Y 559.199,Z 335.832,A -85,B 0,C 180,E1 -3068.674,E2 -3068.674} C_VEL
LIN {X 0,Y 559.212,Z 335.829,A -85,B 0,C 180,E1 -3071.601,E2 -3071.601} C_VEL
LIN {X 0,Y 559.207,Z 335.83,A -85,B 0,C 180,E1 -3074.596,E2 -3074.596} C_VEL
LIN {X 0,Y 559.169,Z 335.834,A -85,B 0,C 180,E1 -3077.557,E2 -3077.557} C_VEL
LIN {X 0,Y 559.172,Z 335.835,A -85,B 0,C 180,E1 -3079.838,E2 -3079.838} C_VEL
LIN {X 0,Y 559.148,Z 335.838,A -85,B 0,C 180,E1 -3082.153,E2 -3082.153} C_VEL
LIN {X 0,Y 559.183,Z 335.832,A -85,B 0,C 180,E1 -3085.298,E2 -3085.298} C_VEL
LIN {X 0,Y 559.188,Z 335.833,A -85,B 0,C 180,E1 -3087.712,E2 -3087.712} C_VEL
LIN {X 0,Y 559.146,Z 335.836,A -85,B 0,C 180,E1 -3090.618,E2 -3090.618} C_VEL
LIN {X 0,Y 558.486,Z 335.921,A -85,B 0,C 180,E1 -3091.22,E2 -3091.22} C_VEL
LIN {X 0,Y 555.627,Z 336.276,A -85,B 0,C 180,E1 -3092.196,E2 -3092.196} C_VEL
LIN {X 0,Y 553.216,Z 336.575,A -85,B 0,C 180,E1 -3092.981,E2 -3092.981} C_VEL
LIN {X 0,Y 552.195,Z 336.705,A -85,B 0,C 180,E1 -3093.588,E2 -3093.588} C_VEL
LIN {X 0,Y 552.12,Z 336.71,A -85,B 0,C 180,E1 -3093.794,E2 -3093.794} C_VEL
LIN {X 0,Y 552.112,Z 336.714,A -85,B 0,C 180,E1 -3096.747,E2 -3096.747} C_VEL
LIN {X 0,Y 552.142,Z 336.71,A -85,B 0,C 180,E1 -3099.527,E2 -3099.527} C_VEL
LIN {X 0,Y 552.136,Z 336.711,A -85,B 0,C 180,E1 -3102.425,E2 -3102.425} C_VEL
LIN {X 0,Y 552.105,Z 336.715,A -85,B 0,C 180,E1 -3105.563,E2 -3105.563} C_VEL
LIN {X 0,Y 552.137,Z 336.71,A -85,B 0,C 180,E1 -3108.677,E2 -3108.677} C_VEL
LIN {X 0,Y 552.122,Z 336.714,A -85,B 0,C 180,E1 -3111.411,E2 -3111.411} C_VEL
LIN {X 0,Y 552.082,Z 336.716,A -85,B 0,C 180,E1 -3114.155,E2 -3114.155} C_VEL
LIN {X 0,Y 552.13,Z 336.711,A -85,B 0,C 180,E1 -3116.815,E2 -3116.815} C_VEL
LIN {X 0,Y 552.106,Z 336.716,A -85,B 0,C 180,E1 -3119.39,E2 -3119.39} C_VEL
LIN {X 0,Y 552.116,Z 336.712,A -85,B 0,C 180,E1 -3121.901,E2 -3121.901} C_VEL
LIN {X 0,Y 552.164,Z 336.707,A -85,B 0,C 180,E1 -3124.649,E2 -3124.649} C_VEL
LIN {X 0,Y 552.1,Z 336.714,A -85,B 0,C 180,E1 -3127.549,E2 -3127.549} C_VEL
LIN {X 0,Y 552.152,Z 336.709,A -85,B 0,C 180,E1 -3130.375,E2 -3130.375} C_VEL
LIN {X 0,Y 552.163,Z 336.708,A -85,B 0,C 180,E1 -3132.977,E2 -3132.977} C_VEL
LIN {X 0,Y 552.142,Z 336.71,A -85,B 0,C 180,E1 -3136.004,E2 -3136.004} C_VEL
LIN {X 0,Y 552.171,Z 336.706,A -85,B 0,C 180,E1 -3138.993,E2 -3138.993} C_VEL
LIN {X 0,Y 552.165,Z 336.708,A -85,B 0,C 180,E1 -3141.951,E2 -3141.951} C_VEL
LIN {X 0,Y 552.23,Z 336.7,A -85,B 0,C 180,E1 -3144.888,E2 -3144.888} C_VEL
LIN {X 0,Y 552.153,Z 336.88,A -85,B 0,C 180,E1 -3145.391,E2 -3145.391} C_VEL
LIN {X 0,Y 552.93,Z 340.954,A -85,B 0,C 180,E1 -3145.534,E2 -3145.534} C_VEL
LIN {X 0,Y 552.811,Z 352.657,A -85,B 0,C 180,E1 -3145.99,E2 -3145.99} C_VEL
LIN {X 0,Y 552.627,Z 364.956,A -85,B 0,C 180,E1 -3146.627,E2 -3146.627} C_VEL
LIN {X 0,Y 552.432,Z 375.956,A -85,B 0,C 180,E1 -3147.356,E2 -3147.356} C_VEL
LIN {X 0,Y 552.267,Z 385.897,A -85,B 0,C 180,E1 -3148.176,E2 -3148.176} C_VEL
LIN {X 0,Y 552.078,Z 394.911,A -85,B 0,C 180,E1 -3149.088,E2 -3149.088} C_VEL
LIN {X 0,Y 551.976,Z 403.716,A -85,B 0,C 180,E1 -3150.182,E2 -3150.182} C_VEL
LIN {X 0,Y 551.827,Z 410.832,A -85,B 0,C 180,E1 -3151.277,E2 -3151.277} C_VEL
LIN {X 0,Y 551.757,Z 417.328,A -85,B 0,C 180,E1 -3152.555,E2 -3152.555} C_VEL
LIN {X 0,Y 551.768,Z 421.639,A -85,B 0,C 180,E1 -3153.651,E2 -3153.651} C_VEL
LIN {X 0,Y 551.722,Z 423.93,A -85,B 0,C 180,E1 -3154.383,E2 -3154.383} C_VEL
LIN {X 0,Y 551.686,Z 425.791,A -85,B 0,C 180,E1 -3155.116,E2 -3155.116} C_VEL
LIN {X 0,Y 551.731,Z 428.087,A -85,B 0,C 180,E1 -3156.496,E2 -3156.496} C_VEL
LIN {X 0,Y 551.693,Z 428.788,A -85,B 0,C 180,E1 -3157.318,E2 -3157.318} C_VEL
LIN {X 0,Y 551.696,Z 429,A -85,B 0,C 180,E1 -3158.055,E2 -3158.055} C_VEL
LIN {X 0,Y 551.671,Z 428.774,A -85,B 0,C 180,E1 -3158.793,E2 -3158.793} C_VEL
LIN {X 0,Y 551.68,Z 427.137,A -85,B 0,C 180,E1 -3160.273,E2 -3160.273} C_VEL
LIN {X 0,Y 551.72,Z 425.177,A -85,B 0,C 180,E1 -3161.227,E2 -3161.227} C_VEL
LIN {X 0,Y 551.749,Z 421.415,A -85,B 0,C 180,E1 -3162.505,E2 -3162.505} C_VEL
LIN {X 0,Y 551.777,Z 416.918,A -85,B 0,C 180,E1 -3163.629,E2 -3163.629} C_VEL
LIN {X 0,Y 551.85,Z 411.159,A -85,B 0,C 180,E1 -3164.756,E2 -3164.756} C_VEL
LIN {X 0,Y 551.938,Z 403.869,A -85,B 0,C 180,E1 -3165.888,E2 -3165.888} C_VEL
LIN {X 0,Y 552.077,Z 394.714,A -85,B 0,C 180,E1 -3167.025,E2 -3167.025} C_VEL
LIN {X 0,Y 552.286,Z 385.243,A -85,B 0,C 180,E1 -3167.974,E2 -3167.974} C_VEL
LIN {X 0,Y 552.444,Z 374.583,A -85,B 0,C 180,E1 -3168.832,E2 -3168.832} C_VEL
LIN {X 0,Y 552.666,Z 363.446,A -85,B 0,C 180,E1 -3169.55,E2 -3169.55} C_VEL
LIN {X 0,Y 552.825,Z 351.063,A -85,B 0,C 180,E1 -3170.171,E2 -3170.171} C_VEL
LIN {X 0,Y 552.802,Z 339.346,A -85,B 0,C 180,E1 -3170.609,E2 -3170.609} C_VEL
LIN {X 0,Y 552.14,Z 336.712,A -85,B 0,C 180,E1 -3170.708,E2 -3170.708} C_VEL
LIN {X 0,Y 552.104,Z 336.716,A -85,B 0,C 180,E1 -3173.576,E2 -3173.576} C_VEL
LIN {X 0,Y 552.133,Z 336.713,A -85,B 0,C 180,E1 -3175.644,E2 -3175.644} C_VEL
LIN {X 0,Y 552.127,Z 336.714,A -85,B 0,C 180,E1 -3178.561,E2 -3178.561} C_VEL
LIN {X 0,Y 552.113,Z 336.715,A -85,B 0,C 180,E1 -3181.475,E2 -3181.475} C_VEL
LIN {X 0,Y 552.135,Z 336.71,A -85,B 0,C 180,E1 -3184.17,E2 -3184.17} C_VEL
LIN {X 0,Y 552.106,Z 336.716,A -85,B 0,C 180,E1 -3186.746,E2 -3186.746} C_VEL
LIN {X 0,Y 552.131,Z 336.713,A -85,B 0,C 180,E1 -3189.526,E2 -3189.526} C_VEL
LIN {X 0,Y 552.132,Z 336.712,A -85,B 0,C 180,E1 -3192.425,E2 -3192.425} C_VEL
LIN {X 0,Y 552.098,Z 336.717,A -85,B 0,C 180,E1 -3195.562,E2 -3195.562} C_VEL
LIN {X 0,Y 552.141,Z 336.711,A -85,B 0,C 180,E1 -3198.675,E2 -3198.675} C_VEL
LIN {X 0,Y 552.12,Z 336.715,A -85,B 0,C 180,E1 -3201.411,E2 -3201.411} C_VEL
LIN {X 0,Y 552.109,Z 336.715,A -85,B 0,C 180,E1 -3204.555,E2 -3204.555} C_VEL
LIN {X 0,Y 552.13,Z 336.711,A -85,B 0,C 180,E1 -3207.15,E2 -3207.15} C_VEL
LIN {X 0,Y 552.145,Z 336.703,A -85,B 0,C 180,E1 -3210.237,E2 -3210.237} C_VEL
LIN {X 0,Y 552.147,Z 336.708,A -85,B 0,C 180,E1 -3212.997,E2 -3212.997} C_VEL
LIN {X 0,Y 552.113,Z 336.714,A -85,B 0,C 180,E1 -3215.161,E2 -3215.161} C_VEL
LIN {X 0,Y 552.096,Z 336.715,A -85,B 0,C 180,E1 -3217.549,E2 -3217.549} C_VEL
LIN {X 0,Y 552.148,Z 336.711,A -85,B 0,C 180,E1 -3220.373,E2 -3220.373} C_VEL
LIN {X 0,Y 552.157,Z 336.706,A -85,B 0,C 180,E1 -3222.977,E2 -3222.977} C_VEL
LIN {X 0,Y 552.136,Z 336.711,A -85,B 0,C 180,E1 -3226.004,E2 -3226.004} C_VEL
LIN {X 0,Y 552.177,Z 336.706,A -85,B 0,C 180,E1 -3228.993,E2 -3228.993} C_VEL
LIN {X 0,Y 552.162,Z 336.707,A -85,B 0,C 180,E1 -3231.951,E2 -3231.951} C_VEL
LIN {X 0,Y 552.231,Z 336.697,A -85,B 0,C 180,E1 -3234.889,E2 -3234.889} C_VEL
LIN {X 0,Y 552.221,Z 336.7,A -85,B 0,C 180,E1 -3237.812,E2 -3237.812} C_VEL
LIN {X 0,Y 552.244,Z 336.696,A -85,B 0,C 180,E1 -3240.729,E2 -3240.729} C_VEL
LIN {X 0,Y 552.207,Z 336.702,A -85,B 0,C 180,E1 -3242.918,E2 -3242.918} C_VEL
LIN {X 0,Y 552.199,Z 336.701,A -85,B 0,C 180,E1 -3245.844,E2 -3245.844} C_VEL
LIN {X 0,Y 552.161,Z 336.707,A -85,B 0,C 180,E1 -3248.786,E2 -3248.786} C_VEL
LIN {X 0,Y 552.16,Z 336.707,A -85,B 0,C 180,E1 -3251.75,E2 -3251.75} C_VEL
LIN {X 0,Y 552.133,Z 336.71,A -85,B 0,C 180,E1 -3254.748,E2 -3254.748} C_VEL
LIN {X 0,Y 552.111,Z 336.712,A -85,B 0,C 180,E1 -3257.788,E2 -3257.788} C_VEL
LIN {X 0,Y 552.128,Z 336.713,A -85,B 0,C 180,E1 -3260.101,E2 -3260.101} C_VEL
LIN {X 0,Y 552.093,Z 336.717,A -85,B 0,C 180,E1 -3262.451,E2 -3262.451} C_VEL
LIN {X 0,Y 552.154,Z 336.71,A -85,B 0,C 180,E1 -3265.351,E2 -3265.351} C_VEL
LIN {X 0,Y 552.125,Z 336.714,A -85,B 0,C 180,E1 -3268.097,E2 -3268.097} C_VEL
LIN {X 0,Y 552.113,Z 336.714,A -85,B 0,C 180,E1 -3270.609,E2 -3270.609} C_VEL
LIN {X 0,Y 552.127,Z 336.714,A -85,B 0,C 180,E1 -3273.185,E2 -3273.185} C_VEL
LIN {X 0,Y 552.112,Z 336.713,A -85,B 0,C 180,E1 -3275.842,E2 -3275.842} C_VEL
LIN {X 0,Y 552.126,Z 336.711,A -85,B 0,C 180,E1 -3279.063,E2 -3279.063} C_VEL
LIN {X 0,Y 552.143,Z 336.708,A -85,B 0,C 180,E1 -3281.444,E2 -3281.444} C_VEL
LIN {X 0,Y 552.095,Z 336.715,A -85,B 0,C 180,E1 -3284.533,E2 -3284.533} C_VEL
LIN {X 0,Y 552.131,Z 336.712,A -85,B 0,C 180,E1 -3287.585,E2 -3287.585} C_VEL
LIN {X 0,Y 552.143,Z 336.711,A -85,B 0,C 180,E1 -3289.793,E2 -3289.793} C_VEL
LIN {X 0,Y 552.186,Z 336.856,A -85,B 0,C 180,E1 -3292.804,E2 -3292.804} C_VEL
LIN {X 0,Y 553.19,Z 343.159,A -85,B 0,C 180,E1 -3294.399,E2 -3294.399} C_VEL
LIN {X 0,Y 552.895,Z 354.525,A -85,B 0,C 180,E1 -3297.029,E2 -3297.029} C_VEL
LIN {X 0,Y 552.783,Z 367.164,A -85,B 0,C 180,E1 -3299.831,E2 -3299.831} C_VEL
LIN {X 0,Y 552.699,Z 380.799,A -85,B 0,C 180,E1 -3302.757,E2 -3302.757} C_VEL
LIN {X 0,Y 552.596,Z 394.456,A -85,B 0,C 180,E1 -3305.586,E2 -3305.586} C_VEL
LIN {X 0,Y 552.502,Z 407.978,A -85,B 0,C 180,E1 -3308.353,E2 -3308.353} C_VEL
LIN {X 0,Y 552.421,Z 419.542,A -85,B 0,C 180,E1 -3310.685,E2 -3310.685} C_VEL
LIN {X 0,Y 552.236,Z 432.253,A -85,B 0,C 180,E1 -3313.361,E2 -3313.361} C_VEL
LIN {X 0,Y 552.064,Z 446.78,A -85,B 0,C 180,E1 -3316.379,E2 -3316.379} C_VEL
LIN {X 0,Y 552.071,Z 449.882,A -85,B 0,C 180,E1 -3316.976,E2 -3316.976} C_VEL
LIN {X 0,Y 553.108,Z 457.255,A -85,B 0,C 180,E1 -3317.129,E2 -3317.129} C_VEL
LIN {X 0,Y 552.976,Z 470.518,A -85,B 0,C 180,E1 -3317.476,E2 -3317.476} C_VEL
LIN {X 0,Y 552.815,Z 482.532,A -85,B 0,C 180,E1 -3317.939,E2 -3317.939} C_VEL
LIN {X 0,Y 552.624,Z 495.124,A -85,B 0,C 180,E1 -3318.592,E2 -3318.592} C_VEL
LIN {X 0,Y 552.426,Z 506.752,A -85,B 0,C 180,E1 -3319.37,E2 -3319.37} C_VEL
LIN {X 0,Y 552.233,Z 517.605,A -85,B 0,C 180,E1 -3320.293,E2 -3320.293} C_VEL
LIN {X 0,Y 552.079,Z 526.418,A -85,B 0,C 180,E1 -3321.214,E2 -3321.214} C_VEL
LIN {X 0,Y 551.949,Z 535.006,A -85,B 0,C 180,E1 -3322.317,E2 -3322.317} C_VEL
LIN {X 0,Y 551.822,Z 541.872,A -85,B 0,C 180,E1 -3323.419,E2 -3323.419} C_VEL
LIN {X 0,Y 551.804,Z 547.368,A -85,B 0,C 180,E1 -3324.519,E2 -3324.519} C_VEL
LIN {X 0,Y 551.764,Z 551.679,A -85,B 0,C 180,E1 -3325.617,E2 -3325.617} C_VEL
LIN {X 0,Y 551.75,Z 553.959,A -85,B 0,C 180,E1 -3326.349,E2 -3326.349} C_VEL
LIN {X 0,Y 551.723,Z 555.809,A -85,B 0,C 180,E1 -3327.08,E2 -3327.08} C_VEL
LIN {X 0,Y 551.645,Z 558.185,A -85,B 0,C 180,E1 -3328.54,E2 -3328.54} C_VEL
LIN {X 0,Y 551.64,Z 559,A -85,B 0,C 180,E1 -3330.001,E2 -3330.001} C_VEL
LIN {X 0,Y 551.645,Z 558.185,A -85,B 0,C 180,E1 -3331.461,E2 -3331.461} C_VEL
LIN {X 0,Y 551.724,Z 555.809,A -85,B 0,C 180,E1 -3332.921,E2 -3332.921} C_VEL
LIN {X 0,Y 551.764,Z 552.894,A -85,B 0,C 180,E1 -3334.018,E2 -3334.018} C_VEL
LIN {X 0,Y 551.724,Z 548.946,A -85,B 0,C 180,E1 -3335.116,E2 -3335.116} C_VEL
LIN {X 0,Y 551.803,Z 543.188,A -85,B 0,C 180,E1 -3336.342,E2 -3336.342} C_VEL
LIN {X 0,Y 551.927,Z 536.233,A -85,B 0,C 180,E1 -3337.5,E2 -3337.5} C_VEL
LIN {X 0,Y 552.083,Z 527.987,A -85,B 0,C 180,E1 -3338.603,E2 -3338.603} C_VEL
LIN {X 0,Y 552.202,Z 519.534,A -85,B 0,C 180,E1 -3339.524,E2 -3339.524} C_VEL
LIN {X 0,Y 552.425,Z 509.088,A -85,B 0,C 180,E1 -3340.445,E2 -3340.445} C_VEL
LIN {X 0,Y 552.6,Z 498.281,A -85,B 0,C 180,E1 -3341.214,E2 -3341.214} C_VEL
LIN {X 0,Y 552.752,Z 487.397,A -85,B 0,C 180,E1 -3341.831,E2 -3341.831} C_VEL
LIN {X 0,Y 552.898,Z 475.749,A -85,B 0,C 180,E1 -3342.34,E2 -3342.34} C_VEL
LIN {X 0,Y 553.045,Z 463.239,A -85,B 0,C 180,E1 -3342.733,E2 -3342.733} C_VEL
LIN {X 0,Y 552.887,Z 454.917,A -85,B 0,C 180,E1 -3342.924,E2 -3342.924} C_VEL
LIN {X 0,Y 552.039,Z 449.612,A -85,B 0,C 180,E1 -3343.037,E2 -3343.037} C_VEL
LIN {X 0,Y 552.174,Z 435.879,A -85,B 0,C 180,E1 -3345.882,E2 -3345.882} C_VEL
LIN {X 0,Y 552.325,Z 424.984,A -85,B 0,C 180,E1 -3348.165,E2 -3348.165} C_VEL
LIN {X 0,Y 552.456,Z 413.866,A -85,B 0,C 180,E1 -3350.478,E2 -3350.478} C_VEL
LIN {X 0,Y 552.591,Z 400.283,A -85,B 0,C 180,E1 -3353.221,E2 -3353.221} C_VEL
LIN {X 0,Y 552.712,Z 384.847,A -85,B 0,C 180,E1 -3356.427,E2 -3356.427} C_VEL
LIN {X 0,Y 552.779,Z 371.296,A -85,B 0,C 180,E1 -3359.307,E2 -3359.307} C_VEL
LIN {X 0,Y 552.868,Z 359.521,A -85,B 0,C 180,E1 -3361.894,E2 -3361.894} C_VEL
LIN {X 0,Y 553.16,Z 346.368,A -85,B 0,C 180,E1 -3364.872,E2 -3364.872} C_VEL
LIN {X 0,Y 553.129,Z 342.542,A -85,B 0,C 180,E1 -3365.766,E2 -3365.766} C_VEL
LIN {X 0,Y 552.151,Z 336.711,A -85,B 0,C 180,E1 -3367.257,E2 -3367.257} C_VEL
LIN {X 0,Y 552.117,Z 336.714,A -85,B 0,C 180,E1 -3370.204,E2 -3370.204} C_VEL
LIN {X 0,Y 552.136,Z 336.711,A -85,B 0,C 180,E1 -3372.426,E2 -3372.426} C_VEL
LIN {X 0,Y 552.103,Z 336.714,A -85,B 0,C 180,E1 -3375.563,E2 -3375.563} C_VEL
LIN {X 0,Y 552.137,Z 336.711,A -85,B 0,C 180,E1 -3378.677,E2 -3378.677} C_VEL
LIN {X 0,Y 552.126,Z 336.712,A -85,B 0,C 180,E1 -3381.412,E2 -3381.412} C_VEL
LIN {X 0,Y 552.091,Z 336.717,A -85,B 0,C 180,E1 -3384.157,E2 -3384.157} C_VEL
LIN {X 0,Y 552.127,Z 336.711,A -85,B 0,C 180,E1 -3386.815,E2 -3386.815} C_VEL
LIN {X 0,Y 552.113,Z 336.714,A -85,B 0,C 180,E1 -3389.391,E2 -3389.391} C_VEL
LIN {X 0,Y 552.115,Z 336.714,A -85,B 0,C 180,E1 -3391.902,E2 -3391.902} C_VEL
LIN {X 0,Y 552.161,Z 336.707,A -85,B 0,C 180,E1 -3394.65,E2 -3394.65} C_VEL
LIN {X 0,Y 552.102,Z 336.716,A -85,B 0,C 180,E1 -3397.55,E2 -3397.55} C_VEL
LIN {X 0,Y 552.156,Z 336.709,A -85,B 0,C 180,E1 -3400.674,E2 -3400.674} C_VEL
LIN {X 0,Y 552.123,Z 336.711,A -85,B 0,C 180,E1 -3403.738,E2 -3403.738} C_VEL
LIN {X 0,Y 552.142,Z 336.709,A -85,B 0,C 180,E1 -3406.005,E2 -3406.005} C_VEL
LIN {X 0,Y 552.167,Z 336.706,A -85,B 0,C 180,E1 -3408.994,E2 -3408.994} C_VEL
LIN {X 0,Y 552.164,Z 336.708,A -85,B 0,C 180,E1 -3411.952,E2 -3411.952} C_VEL
LIN {X 0,Y 552.236,Z 336.697,A -85,B 0,C 180,E1 -3414.889,E2 -3414.889} C_VEL
LIN {X 0,Y 552.224,Z 336.701,A -85,B 0,C 180,E1 -3417.812,E2 -3417.812} C_VEL
LIN {X 0,Y 552.251,Z 336.697,A -85,B 0,C 180,E1 -3420.729,E2 -3420.729} C_VEL
LIN {X 0,Y 552.211,Z 336.701,A -85,B 0,C 180,E1 -3422.918,E2 -3422.918} C_VEL
LIN {X 0,Y 552.202,Z 336.703,A -85,B 0,C 180,E1 -3425.844,E2 -3425.844} C_VEL
LIN {X 0,Y 552.169,Z 336.708,A -85,B 0,C 180,E1 -3428.786,E2 -3428.786} C_VEL
LIN {X 0,Y 552.169,Z 336.706,A -85,B 0,C 180,E1 -3431.751,E2 -3431.751} C_VEL
LIN {X 0,Y 552.144,Z 336.709,A -85,B 0,C 180,E1 -3434.748,E2 -3434.748} C_VEL
LIN {X 0,Y 552.12,Z 336.714,A -85,B 0,C 180,E1 -3437.788,E2 -3437.788} C_VEL
LIN {X 0,Y 552.133,Z 336.713,A -85,B 0,C 180,E1 -3440.101,E2 -3440.101} C_VEL
LIN {X 0,Y 552.099,Z 336.715,A -85,B 0,C 180,E1 -3442.451,E2 -3442.451} C_VEL
LIN {X 0,Y 552.163,Z 336.707,A -85,B 0,C 180,E1 -3445.351,E2 -3445.351} C_VEL
LIN {X 0,Y 552.113,Z 336.714,A -85,B 0,C 180,E1 -3448.099,E2 -3448.099} C_VEL
LIN {X 0,Y 552.109,Z 336.713,A -85,B 0,C 180,E1 -3450.614,E2 -3450.614} C_VEL
LIN {X 0,Y 552.13,Z 336.711,A -85,B 0,C 180,E1 -3453.185,E2 -3453.185} C_VEL
LIN {X 0,Y 552.12,Z 336.71,A -85,B 0,C 180,E1 -3453.794,E2 -3453.794} C_VEL
LIN {X 0,Y 551.482,Z 336.792,A -85,B 0,C 180,E1 -3454.402,E2 -3454.402} C_VEL
LIN {X 0,Y 548.657,Z 337.147,A -85,B 0,C 180,E1 -3455.39,E2 -3455.39} C_VEL
LIN {X 0,Y 546.237,Z 337.449,A -85,B 0,C 180,E1 -3456.185,E2 -3456.185} C_VEL
LIN {X 0,Y 545.169,Z 337.58,A -85,B 0,C 180,E1 -3456.799,E2 -3456.799} C_VEL
LIN {X 0,Y 545.068,Z 337.592,A -85,B 0,C 180,E1 -3457.007,E2 -3457.007} C_VEL
LIN {X 0,Y 545.082,Z 337.591,A -85,B 0,C 180,E1 -3460.142,E2 -3460.142} C_VEL
LIN {X 0,Y 545.085,Z 337.588,A -85,B 0,C 180,E1 -3463.107,E2 -3463.107} C_VEL
LIN {X 0,Y 545.074,Z 337.589,A -85,B 0,C 180,E1 -3466.224,E2 -3466.224} C_VEL
LIN {X 0,Y 545.095,Z 337.587,A -85,B 0,C 180,E1 -3468.886,E2 -3468.886} C_VEL
LIN {X 0,Y 545.056,Z 337.592,A -85,B 0,C 180,E1 -3471.762,E2 -3471.762} C_VEL
LIN {X 0,Y 545.037,Z 337.594,A -85,B 0,C 180,E1 -3474.531,E2 -3474.531} C_VEL
LIN {X 0,Y 545.089,Z 337.59,A -85,B 0,C 180,E1 -3477.212,E2 -3477.212} C_VEL
LIN {X 0,Y 545.068,Z 337.59,A -85,B 0,C 180,E1 -3479.81,E2 -3479.81} C_VEL
LIN {X 0,Y 545.088,Z 337.587,A -85,B 0,C 180,E1 -3482.344,E2 -3482.344} C_VEL
LIN {X 0,Y 545.125,Z 337.585,A -85,B 0,C 180,E1 -3484.82,E2 -3484.82} C_VEL
LIN {X 0,Y 545.046,Z 337.595,A -85,B 0,C 180,E1 -3487.242,E2 -3487.242} C_VEL
LIN {X 0,Y 545.124,Z 337.584,A -85,B 0,C 180,E1 -3490.414,E2 -3490.414} C_VEL
LIN {X 0,Y 545.08,Z 337.589,A -85,B 0,C 180,E1 -3493.521,E2 -3493.521} C_VEL
LIN {X 0,Y 545.102,Z 337.586,A -85,B 0,C 180,E1 -3495.82,E2 -3495.82} C_VEL
LIN {X 0,Y 545.126,Z 337.583,A -85,B 0,C 180,E1 -3498.849,E2 -3498.849} C_VEL
LIN {X 0,Y 545.136,Z 337.584,A -85,B 0,C 180,E1 -3501.847,E2 -3501.847} C_VEL
LIN {X 0,Y 545.205,Z 337.575,A -85,B 0,C 180,E1 -3504.822,E2 -3504.822} C_VEL
LIN {X 0,Y 545.117,Z 337.588,A -85,B 0,C 180,E1 -3505.239,E2 -3505.239} C_VEL
LIN {X 0,Y 545.986,Z 341.312,A -85,B 0,C 180,E1 -3505.385,E2 -3505.385} C_VEL
LIN {X 0,Y 545.854,Z 352.916,A -85,B 0,C 180,E1 -3505.846,E2 -3505.846} C_VEL
LIN {X 0,Y 545.659,Z 365.161,A -85,B 0,C 180,E1 -3506.492,E2 -3506.492} C_VEL
LIN {X 0,Y 545.441,Z 376.125,A -85,B 0,C 180,E1 -3507.23,E2 -3507.23} C_VEL
LIN {X 0,Y 545.215,Z 386.993,A -85,B 0,C 180,E1 -3508.153,E2 -3508.153} C_VEL
LIN {X 0,Y 545.022,Z 395.826,A -85,B 0,C 180,E1 -3509.076,E2 -3509.076} C_VEL
LIN {X 0,Y 544.921,Z 404.474,A -85,B 0,C 180,E1 -3510.184,E2 -3510.184} C_VEL
LIN {X 0,Y 544.734,Z 411.415,A -85,B 0,C 180,E1 -3511.293,E2 -3511.293} C_VEL
LIN {X 0,Y 544.665,Z 417.783,A -85,B 0,C 180,E1 -3512.588,E2 -3512.588} C_VEL
LIN {X 0,Y 544.682,Z 421.99,A -85,B 0,C 180,E1 -3513.698,E2 -3513.698} C_VEL
LIN {X 0,Y 544.617,Z 424.231,A -85,B 0,C 180,E1 -3514.44,E2 -3514.44} C_VEL
LIN {X 0,Y 544.605,Z 426.005,A -85,B 0,C 180,E1 -3515.182,E2 -3515.182} C_VEL
LIN {X 0,Y 544.652,Z 428.295,A -85,B 0,C 180,E1 -3516.668,E2 -3516.668} C_VEL
LIN {X 0,Y 544.605,Z 428.854,A -85,B 0,C 180,E1 -3517.414,E2 -3517.414} C_VEL
LIN {X 0,Y 544.612,Z 428.982,A -85,B 0,C 180,E1 -3518.16,E2 -3518.16} C_VEL
LIN {X 0,Y 544.583,Z 428.038,A -85,B 0,C 180,E1 -3519.658,E2 -3519.658} C_VEL
LIN {X 0,Y 544.585,Z 426.97,A -85,B 0,C 180,E1 -3520.408,E2 -3520.408} C_VEL
LIN {X 0,Y 544.624,Z 425.188,A -85,B 0,C 180,E1 -3521.264,E2 -3521.264} C_VEL
LIN {X 0,Y 544.652,Z 421.056,A -85,B 0,C 180,E1 -3522.671,E2 -3522.671} C_VEL
LIN {X 0,Y 544.717,Z 416.449,A -85,B 0,C 180,E1 -3523.809,E2 -3523.809} C_VEL
LIN {X 0,Y 544.788,Z 410.535,A -85,B 0,C 180,E1 -3524.951,E2 -3524.951} C_VEL
LIN {X 0,Y 544.906,Z 403.08,A -85,B 0,C 180,E1 -3526.099,E2 -3526.099} C_VEL
LIN {X 0,Y 545.077,Z 393.761,A -85,B 0,C 180,E1 -3527.25,E2 -3527.25} C_VEL
LIN {X 0,Y 545.267,Z 383.994,A -85,B 0,C 180,E1 -3528.213,E2 -3528.213} C_VEL
LIN {X 0,Y 545.504,Z 373.072,A -85,B 0,C 180,E1 -3529.081,E2 -3529.081} C_VEL
LIN {X 0,Y 545.726,Z 361.279,A -85,B 0,C 180,E1 -3529.823,E2 -3529.823} C_VEL
LIN {X 0,Y 545.89,Z 349.582,A -85,B 0,C 180,E1 -3530.39,E2 -3530.39} C_VEL
LIN {X 0,Y 545.844,Z 340.486,A -85,B 0,C 180,E1 -3530.736,E2 -3530.736} C_VEL
LIN {X 0,Y 545.109,Z 337.587,A -85,B 0,C 180,E1 -3530.864,E2 -3530.864} C_VEL
LIN {X 0,Y 545.061,Z 337.593,A -85,B 0,C 180,E1 -3533.726,E2 -3533.726} C_VEL
LIN {X 0,Y 545.081,Z 337.59,A -85,B 0,C 180,E1 -3536,E2 -3536} C_VEL
LIN {X 0,Y 545.092,Z 337.59,A -85,B 0,C 180,E1 -3538.747,E2 -3538.747} C_VEL
LIN {X 0,Y 545.061,Z 337.594,A -85,B 0,C 180,E1 -3541.678,E2 -3541.678} C_VEL
LIN {X 0,Y 545.078,Z 337.591,A -85,B 0,C 180,E1 -3544.392,E2 -3544.392} C_VEL
LIN {X 0,Y 545.037,Z 337.596,A -85,B 0,C 180,E1 -3547.303,E2 -3547.303} C_VEL
LIN {X 0,Y 545.067,Z 337.591,A -85,B 0,C 180,E1 -3550.142,E2 -3550.142} C_VEL
LIN {X 0,Y 545.088,Z 337.589,A -85,B 0,C 180,E1 -3553.105,E2 -3553.105} C_VEL
LIN {X 0,Y 545.067,Z 337.592,A -85,B 0,C 180,E1 -3556.224,E2 -3556.224} C_VEL
LIN {X 0,Y 545.102,Z 337.587,A -85,B 0,C 180,E1 -3558.887,E2 -3558.887} C_VEL
LIN {X 0,Y 545.054,Z 337.593,A -85,B 0,C 180,E1 -3561.762,E2 -3561.762} C_VEL
LIN {X 0,Y 545.066,Z 337.593,A -85,B 0,C 180,E1 -3564.533,E2 -3564.533} C_VEL
LIN {X 0,Y 545.082,Z 337.589,A -85,B 0,C 180,E1 -3567.212,E2 -3567.212} C_VEL
LIN {X 0,Y 545.101,Z 337.578,A -85,B 0,C 180,E1 -3569.812,E2 -3569.812} C_VEL
LIN {X 0,Y 545.102,Z 337.585,A -85,B 0,C 180,E1 -3572.824,E2 -3572.824} C_VEL
LIN {X 0,Y 545.052,Z 337.592,A -85,B 0,C 180,E1 -3575.631,E2 -3575.631} C_VEL
LIN {X 0,Y 545.068,Z 337.59,A -85,B 0,C 180,E1 -3578.836,E2 -3578.836} C_VEL
LIN {X 0,Y 545.084,Z 337.589,A -85,B 0,C 180,E1 -3581.195,E2 -3581.195} C_VEL
LIN {X 0,Y 545.077,Z 337.59,A -85,B 0,C 180,E1 -3583.521,E2 -3583.521} C_VEL
LIN {X 0,Y 545.095,Z 337.587,A -85,B 0,C 180,E1 -3585.82,E2 -3585.82} C_VEL
LIN {X 0,Y 545.131,Z 337.583,A -85,B 0,C 180,E1 -3588.849,E2 -3588.849} C_VEL
LIN {X 0,Y 545.132,Z 337.583,A -85,B 0,C 180,E1 -3591.847,E2 -3591.847} C_VEL
LIN {X 0,Y 545.206,Z 337.571,A -85,B 0,C 180,E1 -3594.823,E2 -3594.823} C_VEL
LIN {X 0,Y 545.193,Z 337.575,A -85,B 0,C 180,E1 -3597.783,E2 -3597.783} C_VEL
LIN {X 0,Y 545.214,Z 337.571,A -85,B 0,C 180,E1 -3600.738,E2 -3600.738} C_VEL
LIN {X 0,Y 545.173,Z 337.578,A -85,B 0,C 180,E1 -3602.956,E2 -3602.956} C_VEL
LIN {X 0,Y 545.17,Z 337.577,A -85,B 0,C 180,E1 -3605.919,E2 -3605.919} C_VEL
LIN {X 0,Y 545.119,Z 337.584,A -85,B 0,C 180,E1 -3608.9,E2 -3608.9} C_VEL
LIN {X 0,Y 545.132,Z 337.583,A -85,B 0,C 180,E1 -3611.904,E2 -3611.904} C_VEL
LIN {X 0,Y 545.082,Z 337.589,A -85,B 0,C 180,E1 -3614.944,E2 -3614.944} C_VEL
LIN {X 0,Y 545.079,Z 337.589,A -85,B 0,C 180,E1 -3618.026,E2 -3618.026} C_VEL
LIN {X 0,Y 545.092,Z 337.588,A -85,B 0,C 180,E1 -3620.372,E2 -3620.372} C_VEL
LIN {X 0,Y 545.089,Z 337.588,A -85,B 0,C 180,E1 -3623.559,E2 -3623.559} C_VEL
LIN {X 0,Y 545.086,Z 337.59,A -85,B 0,C 180,E1 -3626,E2 -3626} C_VEL
LIN {X 0,Y 545.09,Z 337.589,A -85,B 0,C 180,E1 -3628.749,E2 -3628.749} C_VEL
LIN {X 0,Y 545.076,Z 337.59,A -85,B 0,C 180,E1 -3631.683,E2 -3631.683} C_VEL
LIN {X 0,Y 545.083,Z 337.589,A -85,B 0,C 180,E1 -3634.563,E2 -3634.563} C_VEL
LIN {X 0,Y 545.069,Z 337.592,A -85,B 0,C 180,E1 -3637.301,E2 -3637.301} C_VEL
LIN {X 0,Y 545.093,Z 337.59,A -85,B 0,C 180,E1 -3640.14,E2 -3640.14} C_VEL
LIN {X 0,Y 545.085,Z 337.591,A -85,B 0,C 180,E1 -3643.106,E2 -3643.106} C_VEL
LIN {X 0,Y 545.066,Z 337.591,A -85,B 0,C 180,E1 -3646.225,E2 -3646.225} C_VEL
LIN {X 0,Y 545.123,Z 337.586,A -85,B 0,C 180,E1 -3648.89,E2 -3648.89} C_VEL
LIN {X 0,Y 545.055,Z 337.595,A -85,B 0,C 180,E1 -3651.764,E2 -3651.764} C_VEL
LIN {X 0,Y 545.096,Z 337.709,A -85,B 0,C 180,E1 -3652.556,E2 -3652.556} C_VEL
LIN {X 0,Y 546.221,Z 343.862,A -85,B 0,C 180,E1 -3654.154,E2 -3654.154} C_VEL
LIN {X 0,Y 546.023,Z 353.288,A -85,B 0,C 180,E1 -3656.396,E2 -3656.396} C_VEL
LIN {X 0,Y 545.798,Z 367.53,A -85,B 0,C 180,E1 -3659.625,E2 -3659.625} C_VEL
LIN {X 0,Y 545.685,Z 380.169,A -85,B 0,C 180,E1 -3662.378,E2 -3662.378} C_VEL
LIN {X 0,Y 545.562,Z 393.736,A -85,B 0,C 180,E1 -3665.25,E2 -3665.25} C_VEL
LIN {X 0,Y 545.462,Z 407.283,A -85,B 0,C 180,E1 -3668.077,E2 -3668.077} C_VEL
LIN {X 0,Y 545.352,Z 420.856,A -85,B 0,C 180,E1 -3670.815,E2 -3670.815} C_VEL
LIN {X 0,Y 545.238,Z 432.253,A -85,B 0,C 180,E1 -3673.141,E2 -3673.141} C_VEL
LIN {X 0,Y 545.018,Z 446.78,A -85,B 0,C 180,E1 -3676.199,E2 -3676.199} C_VEL
LIN {X 0,Y 545.011,Z 449.882,A -85,B 0,C 180,E1 -3676.804,E2 -3676.804} C_VEL
LIN {X 0,Y 546.196,Z 458.394,A -85,B 0,C 180,E1 -3676.987,E2 -3676.987} C_VEL
LIN {X 0,Y 546.057,Z 470.519,A -85,B 0,C 180,E1 -3677.315,E2 -3677.315} C_VEL
LIN {X 0,Y 545.882,Z 482.523,A -85,B 0,C 180,E1 -3677.783,E2 -3677.783} C_VEL
LIN {X 0,Y 545.673,Z 494.044,A -85,B 0,C 180,E1 -3678.381,E2 -3678.381} C_VEL
LIN {X 0,Y 545.486,Z 505.494,A -85,B 0,C 180,E1 -3679.14,E2 -3679.14} C_VEL
LIN {X 0,Y 545.281,Z 515.652,A -85,B 0,C 180,E1 -3679.98,E2 -3679.98} C_VEL
LIN {X 0,Y 545.081,Z 524.791,A -85,B 0,C 180,E1 -3680.913,E2 -3680.913} C_VEL
LIN {X 0,Y 544.916,Z 533.692,A -85,B 0,C 180,E1 -3682.031,E2 -3682.031} C_VEL
LIN {X 0,Y 544.784,Z 540.852,A -85,B 0,C 180,E1 -3683.147,E2 -3683.147} C_VEL
LIN {X 0,Y 544.741,Z 547.368,A -85,B 0,C 180,E1 -3684.448,E2 -3684.448} C_VEL
LIN {X 0,Y 544.66,Z 551.679,A -85,B 0,C 180,E1 -3685.56,E2 -3685.56} C_VEL
LIN {X 0,Y 544.669,Z 553.96,A -85,B 0,C 180,E1 -3686.301,E2 -3686.301} C_VEL
LIN {X 0,Y 544.65,Z 555.809,A -85,B 0,C 180,E1 -3687.042,E2 -3687.042} C_VEL
LIN {X 0,Y 544.546,Z 558.184,A -85,B 0,C 180,E1 -3688.521,E2 -3688.521} C_VEL
LIN {X 0,Y 544.541,Z 559,A -85,B 0,C 180,E1 -3690.001,E2 -3690.001} C_VEL
LIN {X 0,Y 544.546,Z 558.184,A -85,B 0,C 180,E1 -3691.48,E2 -3691.48} C_VEL
LIN {X 0,Y 544.65,Z 555.809,A -85,B 0,C 180,E1 -3692.959,E2 -3692.959} C_VEL
LIN {X 0,Y 544.684,Z 552.894,A -85,B 0,C 180,E1 -3694.07,E2 -3694.07} C_VEL
LIN {X 0,Y 544.654,Z 548.946,A -85,B 0,C 180,E1 -3695.183,E2 -3695.183} C_VEL
LIN {X 0,Y 544.74,Z 543.702,A -85,B 0,C 180,E1 -3696.328,E2 -3696.328} C_VEL
LIN {X 0,Y 544.837,Z 537.464,A -85,B 0,C 180,E1 -3697.412,E2 -3697.412} C_VEL
LIN {X 0,Y 545.007,Z 529.473,A -85,B 0,C 180,E1 -3698.529,E2 -3698.529} C_VEL
LIN {X 0,Y 545.143,Z 521.329,A -85,B 0,C 180,E1 -3699.461,E2 -3699.461} C_VEL
LIN {X 0,Y 545.373,Z 511.392,A -85,B 0,C 180,E1 -3700.394,E2 -3700.394} C_VEL
LIN {X 0,Y 545.566,Z 500.586,A -85,B 0,C 180,E1 -3701.208,E2 -3701.208} C_VEL
LIN {X 0,Y 545.742,Z 489.162,A -85,B 0,C 180,E1 -3701.891,E2 -3701.891} C_VEL
LIN {X 0,Y 545.945,Z 476.961,A -85,B 0,C 180,E1 -3702.453,E2 -3702.453} C_VEL
LIN {X 0,Y 546.102,Z 464.153,A -85,B 0,C 180,E1 -3702.874,E2 -3702.874} C_VEL
LIN {X 0,Y 546.025,Z 456.057,A -85,B 0,C 180,E1 -3703.065,E2 -3703.065} C_VEL
LIN {X 0,Y 545.003,Z 449.612,A -85,B 0,C 180,E1 -3703.209,E2 -3703.209} C_VEL
LIN {X 0,Y 545.146,Z 435.879,A -85,B 0,C 180,E1 -3706.092,E2 -3706.092} C_VEL
LIN {X 0,Y 545.284,Z 426.679,A -85,B 0,C 180,E1 -3708.019,E2 -3708.019} C_VEL
LIN {X 0,Y 545.39,Z 413.095,A -85,B 0,C 180,E1 -3710.755,E2 -3710.755} C_VEL
LIN {X 0,Y 545.524,Z 401.517,A -85,B 0,C 180,E1 -3713.138,E2 -3713.138} C_VEL
LIN {X 0,Y 545.667,Z 386.123,A -85,B 0,C 180,E1 -3716.382,E2 -3716.382} C_VEL
LIN {X 0,Y 545.787,Z 372.617,A -85,B 0,C 180,E1 -3719.296,E2 -3719.296} C_VEL
LIN {X 0,Y 545.906,Z 361.1,A -85,B 0,C 180,E1 -3721.86,E2 -3721.86} C_VEL
LIN {X 0,Y 546.214,Z 347.694,A -85,B 0,C 180,E1 -3724.93,E2 -3724.93} C_VEL
LIN {X 0,Y 546.175,Z 343.857,A -85,B 0,C 180,E1 -3725.839,E2 -3725.839} C_VEL
LIN {X 0,Y 545.086,Z 337.591,A -85,B 0,C 180,E1 -3727.417,E2 -3727.417} C_VEL
LIN {X 0,Y 545.07,Z 337.591,A -85,B 0,C 180,E1 -3730.143,E2 -3730.143} C_VEL
LIN {X 0,Y 545.092,Z 337.589,A -85,B 0,C 180,E1 -3733.106,E2 -3733.106} C_VEL
LIN {X 0,Y 545.055,Z 337.595,A -85,B 0,C 180,E1 -3736.226,E2 -3736.226} C_VEL
LIN {X 0,Y 545.096,Z 337.587,A -85,B 0,C 180,E1 -3738.887,E2 -3738.887} C_VEL
LIN {X 0,Y 545.06,Z 337.593,A -85,B 0,C 180,E1 -3741.763,E2 -3741.763} C_VEL
LIN {X 0,Y 545.042,Z 337.594,A -85,B 0,C 180,E1 -3744.532,E2 -3744.532} C_VEL
LIN {X 0,Y 545.086,Z 337.59,A -85,B 0,C 180,E1 -3747.213,E2 -3747.213} C_VEL
LIN {X 0,Y 545.072,Z 337.591,A -85,B 0,C 180,E1 -3749.811,E2 -3749.811} C_VEL
LIN {X 0,Y 545.086,Z 337.588,A -85,B 0,C 180,E1 -3752.344,E2 -3752.344} C_VEL
LIN {X 0,Y 545.123,Z 337.584,A -85,B 0,C 180,E1 -3754.821,E2 -3754.821} C_VEL
LIN {X 0,Y 545.051,Z 337.594,A -85,B 0,C 180,E1 -3757.243,E2 -3757.243} C_VEL
LIN {X 0,Y 545.122,Z 337.584,A -85,B 0,C 180,E1 -3760.415,E2 -3760.415} C_VEL
LIN {X 0,Y 545.08,Z 337.588,A -85,B 0,C 180,E1 -3763.521,E2 -3763.521} C_VEL
LIN {X 0,Y 545.101,Z 337.586,A -85,B 0,C 180,E1 -3765.82,E2 -3765.82} C_VEL
LIN {X 0,Y 545.123,Z 337.584,A -85,B 0,C 180,E1 -3768.85,E2 -3768.85} C_VEL
LIN {X 0,Y 545.134,Z 337.582,A -85,B 0,C 180,E1 -3771.847,E2 -3771.847} C_VEL
LIN {X 0,Y 545.211,Z 337.572,A -85,B 0,C 180,E1 -3774.823,E2 -3774.823} C_VEL
LIN {X 0,Y 545.197,Z 337.577,A -85,B 0,C 180,E1 -3777.784,E2 -3777.784} C_VEL
LIN {X 0,Y 545.221,Z 337.572,A -85,B 0,C 180,E1 -3780.739,E2 -3780.739} C_VEL
LIN {X 0,Y 545.177,Z 337.577,A -85,B 0,C 180,E1 -3782.956,E2 -3782.956} C_VEL
LIN {X 0,Y 545.174,Z 337.578,A -85,B 0,C 180,E1 -3785.92,E2 -3785.92} C_VEL
LIN {X 0,Y 545.128,Z 337.584,A -85,B 0,C 180,E1 -3788.9,E2 -3788.9} C_VEL
LIN {X 0,Y 545.141,Z 337.582,A -85,B 0,C 180,E1 -3791.904,E2 -3791.904} C_VEL
LIN {X 0,Y 545.093,Z 337.586,A -85,B 0,C 180,E1 -3794.944,E2 -3794.944} C_VEL
LIN {X 0,Y 545.087,Z 337.589,A -85,B 0,C 180,E1 -3798.026,E2 -3798.026} C_VEL
LIN {X 0,Y 545.098,Z 337.587,A -85,B 0,C 180,E1 -3800.372,E2 -3800.372} C_VEL
LIN {X 0,Y 545.095,Z 337.589,A -85,B 0,C 180,E1 -3803.559,E2 -3803.559} C_VEL
LIN {X 0,Y 545.087,Z 337.589,A -85,B 0,C 180,E1 -3806.001,E2 -3806.001} C_VEL
LIN {X 0,Y 545.081,Z 337.589,A -85,B 0,C 180,E1 -3808.745,E2 -3808.745} C_VEL
LIN {X 0,Y 545.066,Z 337.591,A -85,B 0,C 180,E1 -3811.679,E2 -3811.679} C_VEL
LIN {X 0,Y 545.083,Z 337.589,A -85,B 0,C 180,E1 -3814.392,E2 -3814.392} C_VEL
LIN {X 0,Y 545.068,Z 337.592,A -85,B 0,C 180,E1 -3817.007,E2 -3817.007} C_VEL
LIN {X 0,Y 544.363,Z 337.68,A -85,B 0,C 180,E1 -3817.623,E2 -3817.623} C_VEL
LIN {X 0,Y 541.501,Z 338.034,A -85,B 0,C 180,E1 -3818.624,E2 -3818.624} C_VEL
LIN {X 0,Y 539.115,Z 338.333,A -85,B 0,C 180,E1 -3819.43,E2 -3819.43} C_VEL
LIN {X 0,Y 538.105,Z 338.459,A -85,B 0,C 180,E1 -3820.052,E2 -3820.052} C_VEL
LIN {X 0,Y 538.029,Z 338.465,A -85,B 0,C 180,E1 -3820.263,E2 -3820.263} C_VEL
LIN {X 0,Y 538.033,Z 338.467,A -85,B 0,C 180,E1 -3822.987,E2 -3822.987} C_VEL
LIN {X 0,Y 538.037,Z 338.467,A -85,B 0,C 180,E1 -3825.925,E2 -3825.925} C_VEL
LIN {X 0,Y 538.056,Z 338.467,A -85,B 0,C 180,E1 -3829.253,E2 -3829.253} C_VEL
LIN {X 0,Y 537.996,Z 338.471,A -85,B 0,C 180,E1 -3832.122,E2 -3832.122} C_VEL
LIN {X 0,Y 538.002,Z 338.473,A -85,B 0,C 180,E1 -3834.915,E2 -3834.915} C_VEL
LIN {X 0,Y 538.034,Z 338.466,A -85,B 0,C 180,E1 -3837.618,E2 -3837.618} C_VEL
LIN {X 0,Y 538.022,Z 338.468,A -85,B 0,C 180,E1 -3840.239,E2 -3840.239} C_VEL
LIN {X 0,Y 538.064,Z 338.465,A -85,B 0,C 180,E1 -3842.796,E2 -3842.796} C_VEL
LIN {X 0,Y 538.056,Z 338.464,A -85,B 0,C 180,E1 -3845.292,E2 -3845.292} C_VEL
LIN {X 0,Y 538.029,Z 338.469,A -85,B 0,C 180,E1 -3848.546,E2 -3848.546} C_VEL
LIN {X 0,Y 538.041,Z 338.466,A -85,B 0,C 180,E1 -3850.94,E2 -3850.94} C_VEL
LIN {X 0,Y 538.031,Z 338.467,A -85,B 0,C 180,E1 -3853.299,E2 -3853.299} C_VEL
LIN {X 0,Y 538.071,Z 338.461,A -85,B 0,C 180,E1 -3855.63,E2 -3855.63} C_VEL
LIN {X 0,Y 538.085,Z 338.461,A -85,B 0,C 180,E1 -3858.701,E2 -3858.701} C_VEL
LIN {X 0,Y 538.093,Z 338.461,A -85,B 0,C 180,E1 -3861.739,E2 -3861.739} C_VEL
LIN {X 0,Y 538.122,Z 338.458,A -85,B 0,C 180,E1 -3865.036,E2 -3865.036} C_VEL
LIN {X 0,Y 538.111,Z 338.52,A -85,B 0,C 180,E1 -3865.083,E2 -3865.083} C_VEL
LIN {X 0,Y 539.09,Z 343.515,A -85,B 0,C 180,E1 -3865.279,E2 -3865.279} C_VEL
LIN {X 0,Y 538.939,Z 355.625,A -85,B 0,C 180,E1 -3865.793,E2 -3865.793} C_VEL
LIN {X 0,Y 538.692,Z 367.313,A -85,B 0,C 180,E1 -3866.447,E2 -3866.447} C_VEL
LIN {X 0,Y 538.454,Z 377.751,A -85,B 0,C 180,E1 -3867.194,E2 -3867.194} C_VEL
LIN {X 0,Y 538.188,Z 388.224,A -85,B 0,C 180,E1 -3868.129,E2 -3868.129} C_VEL
LIN {X 0,Y 537.967,Z 396.743,A -85,B 0,C 180,E1 -3869.064,E2 -3869.064} C_VEL
LIN {X 0,Y 537.839,Z 405.185,A -85,B 0,C 180,E1 -3870.187,E2 -3870.187} C_VEL
LIN {X 0,Y 537.646,Z 411.983,A -85,B 0,C 180,E1 -3871.31,E2 -3871.31} C_VEL
LIN {X 0,Y 537.58,Z 418.238,A -85,B 0,C 180,E1 -3872.622,E2 -3872.622} C_VEL
LIN {X 0,Y 537.6,Z 422.341,A -85,B 0,C 180,E1 -3873.747,E2 -3873.747} C_VEL
LIN {X 0,Y 537.515,Z 424.513,A -85,B 0,C 180,E1 -3874.499,E2 -3874.499} C_VEL
LIN {X 0,Y 537.526,Z 426.21,A -85,B 0,C 180,E1 -3875.251,E2 -3875.251} C_VEL
LIN {X 0,Y 537.552,Z 428.407,A -85,B 0,C 180,E1 -3876.757,E2 -3876.757} C_VEL
LIN {X 0,Y 537.517,Z 428.893,A -85,B 0,C 180,E1 -3877.512,E2 -3877.512} C_VEL
LIN {X 0,Y 537.507,Z 428.959,A -85,B 0,C 180,E1 -3878.269,E2 -3878.269} C_VEL
LIN {X 0,Y 537.482,Z 427.922,A -85,B 0,C 180,E1 -3879.786,E2 -3879.786} C_VEL
LIN {X 0,Y 537.498,Z 426.772,A -85,B 0,C 180,E1 -3880.547,E2 -3880.547} C_VEL
LIN {X 0,Y 537.539,Z 424.245,A -85,B 0,C 180,E1 -3881.692,E2 -3881.692} C_VEL
LIN {X 0,Y 537.576,Z 420.672,A -85,B 0,C 180,E1 -3882.841,E2 -3882.841} C_VEL
LIN {X 0,Y 537.654,Z 415.938,A -85,B 0,C 180,E1 -3883.994,E2 -3883.994} C_VEL
LIN {X 0,Y 537.749,Z 408.74,A -85,B 0,C 180,E1 -3885.346,E2 -3885.346} C_VEL
LIN {X 0,Y 537.897,Z 400.87,A -85,B 0,C 180,E1 -3886.509,E2 -3886.509} C_VEL
LIN {X 0,Y 538.126,Z 391.348,A -85,B 0,C 180,E1 -3887.639,E2 -3887.639} C_VEL
LIN {X 0,Y 538.331,Z 381.885,A -85,B 0,C 180,E1 -3888.555,E2 -3888.555} C_VEL
LIN {X 0,Y 538.585,Z 371.909,A -85,B 0,C 180,E1 -3889.336,E2 -3889.336} C_VEL
LIN {X 0,Y 538.845,Z 360.264,A -85,B 0,C 180,E1 -3890.058,E2 -3890.058} C_VEL
LIN {X 0,Y 539.021,Z 348.711,A -85,B 0,C 180,E1 -3890.611,E2 -3890.611} C_VEL
LIN {X 0,Y 539.059,Z 342.263,A -85,B 0,C 180,E1 -3890.86,E2 -3890.86} C_VEL
LIN {X 0,Y 538.05,Z 338.466,A -85,B 0,C 180,E1 -3891.013,E2 -3891.013} C_VEL
LIN {X 0,Y 538.008,Z 338.47,A -85,B 0,C 180,E1 -3893.888,E2 -3893.888} C_VEL
LIN {X 0,Y 538.043,Z 338.467,A -85,B 0,C 180,E1 -3896.366,E2 -3896.366} C_VEL
LIN {X 0,Y 538.033,Z 338.468,A -85,B 0,C 180,E1 -3898.933,E2 -3898.933} C_VEL
LIN {X 0,Y 538.016,Z 338.471,A -85,B 0,C 180,E1 -3901.887,E2 -3901.887} C_VEL
LIN {X 0,Y 538.014,Z 338.472,A -85,B 0,C 180,E1 -3904.617,E2 -3904.617} C_VEL
LIN {X 0,Y 538.005,Z 338.472,A -85,B 0,C 180,E1 -3907.169,E2 -3907.169} C_VEL
LIN {X 0,Y 538.024,Z 338.468,A -85,B 0,C 180,E1 -3909.796,E2 -3909.796} C_VEL
LIN {X 0,Y 538.025,Z 338.469,A -85,B 0,C 180,E1 -3912.785,E2 -3912.785} C_VEL
LIN {X 0,Y 538.03,Z 338.468,A -85,B 0,C 180,E1 -3915.925,E2 -3915.925} C_VEL
LIN {X 0,Y 538.078,Z 338.463,A -85,B 0,C 180,E1 -3919.248,E2 -3919.248} C_VEL
LIN {X 0,Y 537.994,Z 338.473,A -85,B 0,C 180,E1 -3922.122,E2 -3922.122} C_VEL
LIN {X 0,Y 538.022,Z 338.469,A -85,B 0,C 180,E1 -3924.917,E2 -3924.917} C_VEL
LIN {X 0,Y 538.031,Z 338.466,A -85,B 0,C 180,E1 -3927.618,E2 -3927.618} C_VEL
LIN {X 0,Y 538.043,Z 338.458,A -85,B 0,C 180,E1 -3930.24,E2 -3930.24} C_VEL
LIN {X 0,Y 538.071,Z 338.461,A -85,B 0,C 180,E1 -3932.796,E2 -3932.796} C_VEL
LIN {X 0,Y 538.049,Z 338.466,A -85,B 0,C 180,E1 -3935.292,E2 -3935.292} C_VEL
LIN {X 0,Y 538.014,Z 338.468,A -85,B 0,C 180,E1 -3938.041,E2 -3938.041} C_VEL
LIN {X 0,Y 538.04,Z 338.465,A -85,B 0,C 180,E1 -3940.94,E2 -3940.94} C_VEL
LIN {X 0,Y 538.028,Z 338.468,A -85,B 0,C 180,E1 -3943.299,E2 -3943.299} C_VEL
LIN {X 0,Y 538.063,Z 338.464,A -85,B 0,C 180,E1 -3945.63,E2 -3945.63} C_VEL
LIN {X 0,Y 538.088,Z 338.46,A -85,B 0,C 180,E1 -3948.702,E2 -3948.702} C_VEL
LIN {X 0,Y 538.089,Z 338.46,A -85,B 0,C 180,E1 -3951.739,E2 -3951.739} C_VEL
LIN {X 0,Y 538.163,Z 338.448,A -85,B 0,C 180,E1 -3954.755,E2 -3954.755} C_VEL
LIN {X 0,Y 538.165,Z 338.451,A -85,B 0,C 180,E1 -3957.755,E2 -3957.755} C_VEL
LIN {X 0,Y 538.184,Z 338.447,A -85,B 0,C 180,E1 -3960.748,E2 -3960.748} C_VEL
LIN {X 0,Y 538.14,Z 338.454,A -85,B 0,C 180,E1 -3962.994,E2 -3962.994} C_VEL
LIN {X 0,Y 538.123,Z 338.455,A -85,B 0,C 180,E1 -3965.997,E2 -3965.997} C_VEL
LIN {X 0,Y 538.07,Z 338.463,A -85,B 0,C 180,E1 -3969.017,E2 -3969.017} C_VEL
LIN {X 0,Y 538.08,Z 338.462,A -85,B 0,C 180,E1 -3972.062,E2 -3972.062} C_VEL
LIN {X 0,Y 538.042,Z 338.467,A -85,B 0,C 180,E1 -3975.144,E2 -3975.144} C_VEL
LIN {X 0,Y 538.031,Z 338.469,A -85,B 0,C 180,E1 -3978.27,E2 -3978.27} C_VEL
LIN {X 0,Y 538.036,Z 338.466,A -85,B 0,C 180,E1 -3980.651,E2 -3980.651} C_VEL
LIN {X 0,Y 538.021,Z 338.468,A -85,B 0,C 180,E1 -3983.888,E2 -3983.888} C_VEL
LIN {X 0,Y 538.048,Z 338.467,A -85,B 0,C 180,E1 -3986.366,E2 -3986.366} C_VEL
LIN {X 0,Y 538.054,Z 338.466,A -85,B 0,C 180,E1 -3988.939,E2 -3988.939} C_VEL
LIN {X 0,Y 538.025,Z 338.469,A -85,B 0,C 180,E1 -3991.891,E2 -3991.891} C_VEL
LIN {X 0,Y 538.032,Z 338.467,A -85,B 0,C 180,E1 -3994.622,E2 -3994.622} C_VEL
LIN {X 0,Y 538.025,Z 338.47,A -85,B 0,C 180,E1 -3997.174,E2 -3997.174} C_VEL
LIN {X 0,Y 538.054,Z 338.465,A -85,B 0,C 180,E1 -3999.794,E2 -3999.794} C_VEL
LIN {X 0,Y 538.022,Z 338.469,A -85,B 0,C 180,E1 -4002.786,E2 -4002.786} C_VEL
LIN {X 0,Y 538.029,Z 338.469,A -85,B 0,C 180,E1 -4005.926,E2 -4005.926} C_VEL
LIN {X 0,Y 538.08,Z 338.464,A -85,B 0,C 180,E1 -4009.249,E2 -4009.249} C_VEL
LIN {X 0,Y 538.024,Z 338.572,A -85,B 0,C 180,E1 -4012.304,E2 -4012.304} C_VEL
LIN {X 0,Y 539.303,Z 345.327,A -85,B 0,C 180,E1 -4014.097,E2 -4014.097} C_VEL
LIN {X 0,Y 539.081,Z 354.341,A -85,B 0,C 180,E1 -4016.277,E2 -4016.277} C_VEL
LIN {X 0,Y 538.852,Z 367.959,A -85,B 0,C 180,E1 -4019.426,E2 -4019.426} C_VEL
LIN {X 0,Y 538.661,Z 380.915,A -85,B 0,C 180,E1 -4022.296,E2 -4022.296} C_VEL
LIN {X 0,Y 538.528,Z 394.95,A -85,B 0,C 180,E1 -4025.317,E2 -4025.317} C_VEL
LIN {X 0,Y 538.405,Z 408.828,A -85,B 0,C 180,E1 -4028.249,E2 -4028.249} C_VEL
LIN {X 0,Y 538.242,Z 421.981,A -85,B 0,C 180,E1 -4030.948,E2 -4030.948} C_VEL
LIN {X 0,Y 538.089,Z 435.533,A -85,B 0,C 180,E1 -4033.692,E2 -4033.692} C_VEL
LIN {X 0,Y 537.992,Z 446.78,A -85,B 0,C 180,E1 -4036.015,E2 -4036.015} C_VEL
LIN {X 0,Y 537.978,Z 449.882,A -85,B 0,C 180,E1 -4036.629,E2 -4036.629} C_VEL
LIN {X 0,Y 539.293,Z 458.394,A -85,B 0,C 180,E1 -4036.818,E2 -4036.818} C_VEL
LIN {X 0,Y 539.119,Z 470.519,A -85,B 0,C 180,E1 -4037.149,E2 -4037.149} C_VEL
LIN {X 0,Y 538.928,Z 482.522,A -85,B 0,C 180,E1 -4037.623,E2 -4037.623} C_VEL
LIN {X 0,Y 538.695,Z 494.693,A -85,B 0,C 180,E1 -4038.267,E2 -4038.267} C_VEL
LIN {X 0,Y 538.511,Z 505.493,A -85,B 0,C 180,E1 -4038.997,E2 -4038.997} C_VEL
LIN {X 0,Y 538.277,Z 515.652,A -85,B 0,C 180,E1 -4039.848,E2 -4039.848} C_VEL
LIN {X 0,Y 538.054,Z 524.79,A -85,B 0,C 180,E1 -4040.793,E2 -4040.793} C_VEL
LIN {X 0,Y 537.85,Z 533.692,A -85,B 0,C 180,E1 -4041.926,E2 -4041.926} C_VEL
LIN {X 0,Y 537.728,Z 540.852,A -85,B 0,C 180,E1 -4043.057,E2 -4043.057} C_VEL
LIN {X 0,Y 537.676,Z 547.368,A -85,B 0,C 180,E1 -4044.375,E2 -4044.375} C_VEL
LIN {X 0,Y 537.557,Z 551.679,A -85,B 0,C 180,E1 -4045.501,E2 -4045.501} C_VEL
LIN {X 0,Y 537.591,Z 553.96,A -85,B 0,C 180,E1 -4046.253,E2 -4046.253} C_VEL
LIN {X 0,Y 537.551,Z 555.808,A -85,B 0,C 180,E1 -4047.003,E2 -4047.003} C_VEL
LIN {X 0,Y 537.452,Z 558.183,A -85,B 0,C 180,E1 -4048.502,E2 -4048.502} C_VEL
LIN {X 0,Y 537.442,Z 559,A -85,B 0,C 180,E1 -4050.001,E2 -4050.001} C_VEL
LIN {X 0,Y 537.452,Z 558.184,A -85,B 0,C 180,E1 -4051.499,E2 -4051.499} C_VEL
LIN {X 0,Y 537.551,Z 555.809,A -85,B 0,C 180,E1 -4052.998,E2 -4052.998} C_VEL
LIN {X 0,Y 537.603,Z 552.894,A -85,B 0,C 180,E1 -4054.124,E2 -4054.124} C_VEL
LIN {X 0,Y 537.587,Z 548.946,A -85,B 0,C 180,E1 -4055.251,E2 -4055.251} C_VEL
LIN {X 0,Y 537.651,Z 544.079,A -85,B 0,C 180,E1 -4056.336,E2 -4056.336} C_VEL
LIN {X 0,Y 537.791,Z 537.463,A -85,B 0,C 180,E1 -4057.51,E2 -4057.51} C_VEL
LIN {X 0,Y 537.973,Z 529.473,A -85,B 0,C 180,E1 -4058.641,E2 -4058.641} C_VEL
LIN {X 0,Y 538.12,Z 521.328,A -85,B 0,C 180,E1 -4059.586,E2 -4059.586} C_VEL
LIN {X 0,Y 538.368,Z 511.391,A -85,B 0,C 180,E1 -4060.531,E2 -4060.531} C_VEL
LIN {X 0,Y 538.576,Z 501.583,A -85,B 0,C 180,E1 -4061.288,E2 -4061.288} C_VEL
LIN {X 0,Y 538.753,Z 490.535,A -85,B 0,C 180,E1 -4061.974,E2 -4061.974} C_VEL
LIN {X 0,Y 538.982,Z 478.089,A -85,B 0,C 180,E1 -4062.568,E2 -4062.568} C_VEL
LIN {X 0,Y 539.175,Z 465.066,A -85,B 0,C 180,E1 -4063.019,E2 -4063.019} C_VEL
LIN {X 0,Y 539.069,Z 456.627,A -85,B 0,C 180,E1 -4063.225,E2 -4063.225} C_VEL
LIN {X 0,Y 537.963,Z 449.612,A -85,B 0,C 180,E1 -4063.385,E2 -4063.385} C_VEL
LIN {X 0,Y 538.076,Z 437.461,A -85,B 0,C 180,E1 -4065.92,E2 -4065.92} C_VEL
LIN {X 0,Y 538.209,Z 425.919,A -85,B 0,C 180,E1 -4068.264,E2 -4068.264} C_VEL
LIN {X 0,Y 538.348,Z 412.326,A -85,B 0,C 180,E1 -4071.04,E2 -4071.04} C_VEL
LIN {X 0,Y 538.5,Z 398.31,A -85,B 0,C 180,E1 -4073.996,E2 -4073.996} C_VEL
LIN {X 0,Y 538.651,Z 385.445,A -85,B 0,C 180,E1 -4076.753,E2 -4076.753} C_VEL
LIN {X 0,Y 538.805,Z 372.009,A -85,B 0,C 180,E1 -4079.714,E2 -4079.714} C_VEL
LIN {X 0,Y 538.962,Z 360.49,A -85,B 0,C 180,E1 -4082.32,E2 -4082.32} C_VEL
LIN {X 0,Y 539.281,Z 348.999,A -85,B 0,C 180,E1 -4084.989,E2 -4084.989} C_VEL
LIN {X 0,Y 539.113,Z 344.513,A -85,B 0,C 180,E1 -4086.075,E2 -4086.075} C_VEL
LIN {X 0,Y 538.037,Z 338.468,A -85,B 0,C 180,E1 -4087.648,E2 -4087.648} C_VEL
LIN {X 0,Y 538.054,Z 338.466,A -85,B 0,C 180,E1 -4090.776,E2 -4090.776} C_VEL
LIN {X 0,Y 538.035,Z 338.469,A -85,B 0,C 180,E1 -4094.075,E2 -4094.075} C_VEL
LIN {X 0,Y 538.024,Z 338.471,A -85,B 0,C 180,E1 -4097.214,E2 -4097.214} C_VEL
LIN {X 0,Y 538.035,Z 338.465,A -85,B 0,C 180,E1 -4100.204,E2 -4100.204} C_VEL
LIN {X 0,Y 538.03,Z 338.468,A -85,B 0,C 180,E1 -4103.067,E2 -4103.067} C_VEL
LIN {X 0,Y 538.025,Z 338.467,A -85,B 0,C 180,E1 -4105.827,E2 -4105.827} C_VEL
LIN {X 0,Y 538.03,Z 338.469,A -85,B 0,C 180,E1 -4108.5,E2 -4108.5} C_VEL
LIN {X 0,Y 538.065,Z 338.463,A -85,B 0,C 180,E1 -4111.1,E2 -4111.1} C_VEL
LIN {X 0,Y 538.046,Z 338.464,A -85,B 0,C 180,E1 -4113.634,E2 -4113.634} C_VEL
LIN {X 0,Y 538.029,Z 338.467,A -85,B 0,C 180,E1 -4116.118,E2 -4116.118} C_VEL
LIN {X 0,Y 538.043,Z 338.466,A -85,B 0,C 180,E1 -4119.349,E2 -4119.349} C_VEL
LIN {X 0,Y 538.041,Z 338.466,A -85,B 0,C 180,E1 -4122.468,E2 -4122.468} C_VEL
LIN {X 0,Y 538.07,Z 338.462,A -85,B 0,C 180,E1 -4125.631,E2 -4125.631} C_VEL
LIN {X 0,Y 538.083,Z 338.463,A -85,B 0,C 180,E1 -4128.702,E2 -4128.702} C_VEL
LIN {X 0,Y 538.091,Z 338.459,A -85,B 0,C 180,E1 -4131.74,E2 -4131.74} C_VEL
LIN {X 0,Y 538.169,Z 338.45,A -85,B 0,C 180,E1 -4134.755,E2 -4134.755} C_VEL
LIN {X 0,Y 538.169,Z 338.452,A -85,B 0,C 180,E1 -4137.755,E2 -4137.755} C_VEL
LIN {X 0,Y 538.191,Z 338.448,A -85,B 0,C 180,E1 -4140.748,E2 -4140.748} C_VEL
LIN {X 0,Y 538.144,Z 338.454,A -85,B 0,C 180,E1 -4142.995,E2 -4142.995} C_VEL
LIN {X 0,Y 538.128,Z 338.455,A -85,B 0,C 180,E1 -4145.997,E2 -4145.997} C_VEL
LIN {X 0,Y 538.078,Z 338.462,A -85,B 0,C 180,E1 -4149.018,E2 -4149.018} C_VEL
LIN {X 0,Y 538.09,Z 338.461,A -85,B 0,C 180,E1 -4152.063,E2 -4152.063} C_VEL
LIN {X 0,Y 538.053,Z 338.463,A -85,B 0,C 180,E1 -4155.144,E2 -4155.144} C_VEL
LIN {X 0,Y 538.039,Z 338.466,A -85,B 0,C 180,E1 -4158.27,E2 -4158.27} C_VEL
LIN {X 0,Y 538.044,Z 338.465,A -85,B 0,C 180,E1 -4160.651,E2 -4160.651} C_VEL
LIN {X 0,Y 538.032,Z 338.467,A -85,B 0,C 180,E1 -4163.887,E2 -4163.887} C_VEL
LIN {X 0,Y 538.049,Z 338.465,A -85,B 0,C 180,E1 -4166.367,E2 -4166.367} C_VEL
LIN {X 0,Y 538.036,Z 338.467,A -85,B 0,C 180,E1 -4168.933,E2 -4168.933} C_VEL
LIN {X 0,Y 538.021,Z 338.468,A -85,B 0,C 180,E1 -4171.888,E2 -4171.888} C_VEL
LIN {X 0,Y 538.02,Z 338.469,A -85,B 0,C 180,E1 -4174.618,E2 -4174.618} C_VEL
LIN {X 0,Y 538.011,Z 338.471,A -85,B 0,C 180,E1 -4177.17,E2 -4177.17} C_VEL
LIN {X 0,Y 538.029,Z 338.465,A -85,B 0,C 180,E1 -4180.263,E2 -4180.263} C_VEL
LIN {X 0,Y 537.377,Z 338.549,A -85,B 0,C 180,E1 -4180.888,E2 -4180.888} C_VEL
LIN {X 0,Y 534.521,Z 338.909,A -85,B 0,C 180,E1 -4181.903,E2 -4181.903} C_VEL
LIN {X 0,Y 532.093,Z 339.212,A -85,B 0,C 180,E1 -4182.72,E2 -4182.72} C_VEL
LIN {X 0,Y 531.046,Z 339.34,A -85,B 0,C 180,E1 -4183.351,E2 -4183.351} C_VEL
LIN {X 0,Y 530.959,Z 339.349,A -85,B 0,C 180,E1 -4183.565,E2 -4183.565} C_VEL
LIN {X 0,Y 530.972,Z 339.345,A -85,B 0,C 180,E1 -4186.505,E2 -4186.505} C_VEL
LIN {X 0,Y 530.993,Z 339.344,A -85,B 0,C 180,E1 -4188.976,E2 -4188.976} C_VEL
LIN {X 0,Y 530.961,Z 339.349,A -85,B 0,C 180,E1 -4191.529,E2 -4191.529} C_VEL
LIN {X 0,Y 530.957,Z 339.347,A -85,B 0,C 180,E1 -4194.38,E2 -4194.38} C_VEL
LIN {X 0,Y 530.977,Z 339.348,A -85,B 0,C 180,E1 -4197.133,E2 -4197.133} C_VEL
LIN {X 0,Y 530.968,Z 339.346,A -85,B 0,C 180,E1 -4199.802,E2 -4199.802} C_VEL
LIN {X 0,Y 531.02,Z 339.34,A -85,B 0,C 180,E1 -4202.467,E2 -4202.467} C_VEL
LIN {X 0,Y 531.013,Z 339.344,A -85,B 0,C 180,E1 -4204.942,E2 -4204.942} C_VEL
LIN {X 0,Y 530.979,Z 339.346,A -85,B 0,C 180,E1 -4208.246,E2 -4208.246} C_VEL
LIN {X 0,Y 531.001,Z 339.345,A -85,B 0,C 180,E1 -4210.677,E2 -4210.677} C_VEL
LIN {X 0,Y 530.993,Z 339.344,A -85,B 0,C 180,E1 -4213.071,E2 -4213.071} C_VEL
LIN {X 0,Y 531.027,Z 339.339,A -85,B 0,C 180,E1 -4215.436,E2 -4215.436} C_VEL
LIN {X 0,Y 531.045,Z 339.339,A -85,B 0,C 180,E1 -4218.549,E2 -4218.549} C_VEL
LIN {X 0,Y 531.063,Z 339.336,A -85,B 0,C 180,E1 -4221.629,E2 -4221.629} C_VEL
LIN {X 0,Y 531.11,Z 339.331,A -85,B 0,C 180,E1 -4224.899,E2 -4224.899} C_VEL
LIN {X 0,Y 532.211,Z 344.684,A -85,B 0,C 180,E1 -4225.123,E2 -4225.123} C_VEL
LIN {X 0,Y 532.058,Z 356.715,A -85,B 0,C 180,E1 -4225.644,E2 -4225.644} C_VEL
LIN {X 0,Y 531.799,Z 368.344,A -85,B 0,C 180,E1 -4226.306,E2 -4226.306} C_VEL
LIN {X 0,Y 531.511,Z 379.888,A -85,B 0,C 180,E1 -4227.157,E2 -4227.157} C_VEL
LIN {X 0,Y 531.232,Z 390.146,A -85,B 0,C 180,E1 -4228.104,E2 -4228.104} C_VEL
LIN {X 0,Y 531.01,Z 398.473,A -85,B 0,C 180,E1 -4229.052,E2 -4229.052} C_VEL
LIN {X 0,Y 530.839,Z 406.564,A -85,B 0,C 180,E1 -4230.189,E2 -4230.189} C_VEL
LIN {X 0,Y 530.663,Z 412.13,A -85,B 0,C 180,E1 -4231.138,E2 -4231.138} C_VEL
LIN {X 0,Y 530.5,Z 417.56,A -85,B 0,C 180,E1 -4232.277,E2 -4232.277} C_VEL
LIN {X 0,Y 530.551,Z 421.806,A -85,B 0,C 180,E1 -4233.417,E2 -4233.417} C_VEL
LIN {X 0,Y 530.424,Z 425.052,A -85,B 0,C 180,E1 -4234.559,E2 -4234.559} C_VEL
LIN {X 0,Y 530.448,Z 426.652,A -85,B 0,C 180,E1 -4235.321,E2 -4235.321} C_VEL
LIN {X 0,Y 530.468,Z 428.687,A -85,B 0,C 180,E1 -4236.848,E2 -4236.848} C_VEL
LIN {X 0,Y 530.417,Z 429.11,A -85,B 0,C 180,E1 -4238.38,E2 -4238.38} C_VEL
LIN {X 0,Y 530.363,Z 428.759,A -85,B 0,C 180,E1 -4239.149,E2 -4239.149} C_VEL
LIN {X 0,Y 530.392,Z 428,A -85,B 0,C 180,E1 -4239.919,E2 -4239.919} C_VEL
LIN {X 0,Y 530.479,Z 425.423,A -85,B 0,C 180,E1 -4241.365,E2 -4241.365} C_VEL
LIN {X 0,Y 530.482,Z 421.972,A -85,B 0,C 180,E1 -4242.626,E2 -4242.626} C_VEL
LIN {X 0,Y 530.578,Z 417.639,A -85,B 0,C 180,E1 -4243.793,E2 -4243.793} C_VEL
LIN {X 0,Y 530.685,Z 412.007,A -85,B 0,C 180,E1 -4244.978,E2 -4244.978} C_VEL
LIN {X 0,Y 530.846,Z 405.034,A -85,B 0,C 180,E1 -4246.142,E2 -4246.142} C_VEL
LIN {X 0,Y 531.077,Z 396.313,A -85,B 0,C 180,E1 -4247.301,E2 -4247.301} C_VEL
LIN {X 0,Y 531.346,Z 386.937,A -85,B 0,C 180,E1 -4248.308,E2 -4248.308} C_VEL
LIN {X 0,Y 531.585,Z 376.604,A -85,B 0,C 180,E1 -4249.2,E2 -4249.2} C_VEL
LIN {X 0,Y 531.871,Z 365.01,A -85,B 0,C 180,E1 -4249.992,E2 -4249.992} C_VEL
LIN {X 0,Y 532.1,Z 352.996,A -85,B 0,C 180,E1 -4250.63,E2 -4250.63} C_VEL
LIN {X 0,Y 532.248,Z 344.174,A -85,B 0,C 180,E1 -4250.987,E2 -4250.987} C_VEL
LIN {X 0,Y 531.01,Z 339.343,A -85,B 0,C 180,E1 -4251.191,E2 -4251.191} C_VEL
LIN {X 0,Y 530.975,Z 339.346,A -85,B 0,C 180,E1 -4254.224,E2 -4254.224} C_VEL
LIN {X 0,Y 531.002,Z 339.345,A -85,B 0,C 180,E1 -4256.743,E2 -4256.743} C_VEL
LIN {X 0,Y 530.984,Z 339.347,A -85,B 0,C 180,E1 -4259.322,E2 -4259.322} C_VEL
LIN {X 0,Y 530.972,Z 339.348,A -85,B 0,C 180,E1 -4262.1,E2 -4262.1} C_VEL
LIN {X 0,Y 530.972,Z 339.348,A -85,B 0,C 180,E1 -4264.851,E2 -4264.851} C_VEL
LIN {X 0,Y 530.966,Z 339.35,A -85,B 0,C 180,E1 -4267.507,E2 -4267.507} C_VEL
LIN {X 0,Y 530.982,Z 339.347,A -85,B 0,C 180,E1 -4270.432,E2 -4270.432} C_VEL
LIN {X 0,Y 530.967,Z 339.349,A -85,B 0,C 180,E1 -4273.494,E2 -4273.494} C_VEL
LIN {X 0,Y 530.965,Z 339.349,A -85,B 0,C 180,E1 -4276.505,E2 -4276.505} C_VEL
LIN {X 0,Y 531.026,Z 339.341,A -85,B 0,C 180,E1 -4279.571,E2 -4279.571} C_VEL
LIN {X 0,Y 530.969,Z 339.348,A -85,B 0,C 180,E1 -4282.576,E2 -4282.576} C_VEL
LIN {X 0,Y 531.004,Z 339.344,A -85,B 0,C 180,E1 -4285.311,E2 -4285.311} C_VEL
LIN {X 0,Y 530.982,Z 339.343,A -85,B 0,C 180,E1 -4288.032,E2 -4288.032} C_VEL
LIN {X 0,Y 531.006,Z 339.336,A -85,B 0,C 180,E1 -4290.87,E2 -4290.87} C_VEL
LIN {X 0,Y 531.012,Z 339.341,A -85,B 0,C 180,E1 -4293.256,E2 -4293.256} C_VEL
LIN {X 0,Y 530.995,Z 339.342,A -85,B 0,C 180,E1 -4295.957,E2 -4295.957} C_VEL
LIN {X 0,Y 531.001,Z 339.343,A -85,B 0,C 180,E1 -4299.062,E2 -4299.062} C_VEL
LIN {X 0,Y 531.015,Z 339.34,A -85,B 0,C 180,E1 -4302.277,E2 -4302.277} C_VEL
LIN {X 0,Y 531.039,Z 339.34,A -85,B 0,C 180,E1 -4305.436,E2 -4305.436} C_VEL
LIN {X 0,Y 531.057,Z 339.337,A -85,B 0,C 180,E1 -4308.55,E2 -4308.55} C_VEL
LIN {X 0,Y 531.058,Z 339.336,A -85,B 0,C 180,E1 -4311.629,E2 -4311.629} C_VEL
LIN {X 0,Y 531.122,Z 339.325,A -85,B 0,C 180,E1 -4314.685,E2 -4314.685} C_VEL
LIN {X 0,Y 531.137,Z 339.326,A -85,B 0,C 180,E1 -4317.725,E2 -4317.725} C_VEL
LIN {X 0,Y 531.154,Z 339.322,A -85,B 0,C 180,E1 -4320.758,E2 -4320.758} C_VEL
LIN {X 0,Y 531.106,Z 339.331,A -85,B 0,C 180,E1 -4323.034,E2 -4323.034} C_VEL
LIN {X 0,Y 531.083,Z 339.332,A -85,B 0,C 180,E1 -4326.077,E2 -4326.077} C_VEL
LIN {X 0,Y 531.03,Z 339.34,A -85,B 0,C 180,E1 -4329.138,E2 -4329.138} C_VEL
LIN {X 0,Y 531.038,Z 339.34,A -85,B 0,C 180,E1 -4332.225,E2 -4332.225} C_VEL
LIN {X 0,Y 530.993,Z 339.346,A -85,B 0,C 180,E1 -4335.35,E2 -4335.35} C_VEL
LIN {X 0,Y 531.013,Z 339.34,A -85,B 0,C 180,E1 -4337.722,E2 -4337.722} C_VEL
LIN {X 0,Y 530.997,Z 339.343,A -85,B 0,C 180,E1 -4340.938,E2 -4340.938} C_VEL
LIN {X 0,Y 530.977,Z 339.348,A -85,B 0,C 180,E1 -4344.225,E2 -4344.225} C_VEL
LIN {X 0,Y 531.01,Z 339.343,A -85,B 0,C 180,E1 -4346.743,E2 -4346.743} C_VEL
LIN {X 0,Y 530.998,Z 339.345,A -85,B 0,C 180,E1 -4349.322,E2 -4349.322} C_VEL
LIN {X 0,Y 530.978,Z 339.348,A -85,B 0,C 180,E1 -4352.103,E2 -4352.103} C_VEL
LIN {X 0,Y 530.989,Z 339.345,A -85,B 0,C 180,E1 -4354.855,E2 -4354.855} C_VEL
LIN {X 0,Y 530.972,Z 339.346,A -85,B 0,C 180,E1 -4357.507,E2 -4357.507} C_VEL
LIN {X 0,Y 531.025,Z 339.341,A -85,B 0,C 180,E1 -4360.429,E2 -4360.429} C_VEL
LIN {X 0,Y 530.965,Z 339.348,A -85,B 0,C 180,E1 -4363.495,E2 -4363.495} C_VEL
LIN {X 0,Y 530.967,Z 339.346,A -85,B 0,C 180,E1 -4366.506,E2 -4366.506} C_VEL
LIN {X 0,Y 531.027,Z 339.342,A -85,B 0,C 180,E1 -4369.572,E2 -4369.572} C_VEL
LIN {X 0,Y 530.996,Z 339.54,A -85,B 0,C 180,E1 -4372.076,E2 -4372.076} C_VEL
LIN {X 0,Y 532.391,Z 346.994,A -85,B 0,C 180,E1 -4374.09,E2 -4374.09} C_VEL
LIN {X 0,Y 532.134,Z 356.05,A -85,B 0,C 180,E1 -4376.31,E2 -4376.31} C_VEL
LIN {X 0,Y 531.841,Z 369.741,A -85,B 0,C 180,E1 -4379.526,E2 -4379.526} C_VEL
LIN {X 0,Y 531.635,Z 382.682,A -85,B 0,C 180,E1 -4382.44,E2 -4382.44} C_VEL
LIN {X 0,Y 531.486,Z 396.174,A -85,B 0,C 180,E1 -4385.385,E2 -4385.385} C_VEL
LIN {X 0,Y 531.285,Z 411.521,A -85,B 0,C 180,E1 -4388.668,E2 -4388.668} C_VEL
LIN {X 0,Y 531.147,Z 423.107,A -85,B 0,C 180,E1 -4391.085,E2 -4391.085} C_VEL
LIN {X 0,Y 531.045,Z 434.729,A -85,B 0,C 180,E1 -4393.469,E2 -4393.469} C_VEL
LIN {X 0,Y 530.856,Z 449.305,A -85,B 0,C 180,E1 -4396.446,E2 -4396.446} C_VEL
LIN {X 0,Y 532.345,Z 460.233,A -85,B 0,C 180,E1 -4396.691,E2 -4396.691} C_VEL
LIN {X 0,Y 532.157,Z 472.977,A -85,B 0,C 180,E1 -4397.075,E2 -4397.075} C_VEL
LIN {X 0,Y 531.928,Z 485.412,A -85,B 0,C 180,E1 -4397.603,E2 -4397.603} C_VEL
LIN {X 0,Y 531.697,Z 496.966,A -85,B 0,C 180,E1 -4398.251,E2 -4398.251} C_VEL
LIN {X 0,Y 531.433,Z 507.924,A -85,B 0,C 180,E1 -4399.042,E2 -4399.042} C_VEL
LIN {X 0,Y 531.194,Z 517.603,A -85,B 0,C 180,E1 -4399.904,E2 -4399.904} C_VEL
LIN {X 0,Y 530.969,Z 526.417,A -85,B 0,C 180,E1 -4400.861,E2 -4400.861} C_VEL
LIN {X 0,Y 530.779,Z 535.007,A -85,B 0,C 180,E1 -4402.009,E2 -4402.009} C_VEL
LIN {X 0,Y 530.636,Z 541.871,A -85,B 0,C 180,E1 -4403.155,E2 -4403.155} C_VEL
LIN {X 0,Y 530.611,Z 547.368,A -85,B 0,C 180,E1 -4404.299,E2 -4404.299} C_VEL
LIN {X 0,Y 530.457,Z 551.678,A -85,B 0,C 180,E1 -4405.441,E2 -4405.441} C_VEL
LIN {X 0,Y 530.516,Z 553.959,A -85,B 0,C 180,E1 -4406.203,E2 -4406.203} C_VEL
LIN {X 0,Y 530.457,Z 555.808,A -85,B 0,C 180,E1 -4406.963,E2 -4406.963} C_VEL
LIN {X 0,Y 530.411,Z 557.194,A -85,B 0,C 180,E1 -4407.722,E2 -4407.722} C_VEL
LIN {X 0,Y 530.344,Z 558.786,A -85,B 0,C 180,E1 -4409.241,E2 -4409.241} C_VEL
LIN {X 0,Y 530.342,Z 559,A -85,B 0,C 180,E1 -4410.001,E2 -4410.001} C_VEL
LIN {X 0,Y 530.361,Z 558.183,A -85,B 0,C 180,E1 -4411.519,E2 -4411.519} C_VEL
LIN {X 0,Y 530.411,Z 557.195,A -85,B 0,C 180,E1 -4412.279,E2 -4412.279} C_VEL
LIN {X 0,Y 530.457,Z 555.809,A -85,B 0,C 180,E1 -4413.038,E2 -4413.038} C_VEL
LIN {X 0,Y 530.522,Z 552.894,A -85,B 0,C 180,E1 -4414.179,E2 -4414.179} C_VEL
LIN {X 0,Y 530.525,Z 548.946,A -85,B 0,C 180,E1 -4415.321,E2 -4415.321} C_VEL
LIN {X 0,Y 530.599,Z 543.26,A -85,B 0,C 180,E1 -4416.582,E2 -4416.582} C_VEL
LIN {X 0,Y 530.758,Z 536.232,A -85,B 0,C 180,E1 -4417.801,E2 -4417.801} C_VEL
LIN {X 0,Y 530.931,Z 527.988,A -85,B 0,C 180,E1 -4418.948,E2 -4418.948} C_VEL
LIN {X 0,Y 531.119,Z 519.534,A -85,B 0,C 180,E1 -4419.906,E2 -4419.906} C_VEL
LIN {X 0,Y 531.422,Z 509.083,A -85,B 0,C 180,E1 -4420.863,E2 -4420.863} C_VEL
LIN {X 0,Y 531.693,Z 498.348,A -85,B 0,C 180,E1 -4421.656,E2 -4421.656} C_VEL
LIN {X 0,Y 531.909,Z 487.332,A -85,B 0,C 180,E1 -4422.302,E2 -4422.302} C_VEL
LIN {X 0,Y 532.107,Z 475.559,A -85,B 0,C 180,E1 -4422.83,E2 -4422.83} C_VEL
LIN {X 0,Y 532.314,Z 462.03,A -85,B 0,C 180,E1 -4423.262,E2 -4423.262} C_VEL
LIN {X 0,Y 532.078,Z 457.148,A -85,B 0,C 180,E1 -4423.383,E2 -4423.383} C_VEL
LIN {X 0,Y 530.866,Z 449.236,A -85,B 0,C 180,E1 -4423.567,E2 -4423.567} C_VEL
LIN {X 0,Y 531.047,Z 434.794,A -85,B 0,C 180,E1 -4426.532,E2 -4426.532} C_VEL
LIN {X 0,Y 531.214,Z 421.288,A -85,B 0,C 180,E1 -4429.315,E2 -4429.315} C_VEL
LIN {X 0,Y 531.374,Z 407.518,A -85,B 0,C 180,E1 -4432.206,E2 -4432.206} C_VEL
LIN {X 0,Y 531.492,Z 394.379,A -85,B 0,C 180,E1 -4435.034,E2 -4435.034} C_VEL
LIN {X 0,Y 531.712,Z 380.921,A -85,B 0,C 180,E1 -4437.996,E2 -4437.996} C_VEL
LIN {X 0,Y 531.9,Z 367.538,A -85,B 0,C 180,E1 -4441.019,E2 -4441.019} C_VEL
LIN {X 0,Y 532.184,Z 354.11,A -85,B 0,C 180,E1 -4444.143,E2 -4444.143} C_VEL
LIN {X 0,Y 532.28,Z 346.78,A -85,B 0,C 180,E1 -4445.908,E2 -4445.908} C_VEL
LIN {X 0,Y 530.966,Z 339.349,A -85,B 0,C 180,E1 -4447.868,E2 -4447.868} C_VEL
LIN {X 0,Y 530.986,Z 339.347,A -85,B 0,C 180,E1 -4450.433,E2 -4450.433} C_VEL
LIN {X 0,Y 530.976,Z 339.347,A -85,B 0,C 180,E1 -4453.283,E2 -4453.283} C_VEL
LIN {X 0,Y 530.989,Z 339.344,A -85,B 0,C 180,E1 -4455.622,E2 -4455.622} C_VEL
LIN {X 0,Y 531.001,Z 339.345,A -85,B 0,C 180,E1 -4458.565,E2 -4458.565} C_VEL
LIN {X 0,Y 530.965,Z 339.348,A -85,B 0,C 180,E1 -4461.53,E2 -4461.53} C_VEL
LIN {X 0,Y 530.959,Z 339.348,A -85,B 0,C 180,E1 -4464.38,E2 -4464.38} C_VEL
LIN {X 0,Y 530.977,Z 339.347,A -85,B 0,C 180,E1 -4467.134,E2 -4467.134} C_VEL
LIN {X 0,Y 530.975,Z 339.346,A -85,B 0,C 180,E1 -4469.803,E2 -4469.803} C_VEL
LIN {X 0,Y 531.018,Z 339.341,A -85,B 0,C 180,E1 -4472.468,E2 -4472.468} C_VEL
LIN {X 0,Y 531.011,Z 339.343,A -85,B 0,C 180,E1 -4474.943,E2 -4474.943} C_VEL
LIN {X 0,Y 530.977,Z 339.346,A -85,B 0,C 180,E1 -4478.247,E2 -4478.247} C_VEL
LIN {X 0,Y 530.997,Z 339.345,A -85,B 0,C 180,E1 -4480.677,E2 -4480.677} C_VEL
LIN {X 0,Y 530.981,Z 339.347,A -85,B 0,C 180,E1 -4483.071,E2 -4483.071} C_VEL
LIN {X 0,Y 531.025,Z 339.34,A -85,B 0,C 180,E1 -4485.436,E2 -4485.436} C_VEL
LIN {X 0,Y 531.042,Z 339.34,A -85,B 0,C 180,E1 -4488.55,E2 -4488.55} C_VEL
LIN {X 0,Y 531.06,Z 339.334,A -85,B 0,C 180,E1 -4491.63,E2 -4491.63} C_VEL
LIN {X 0,Y 531.128,Z 339.327,A -85,B 0,C 180,E1 -4494.685,E2 -4494.685} C_VEL
LIN {X 0,Y 531.142,Z 339.327,A -85,B 0,C 180,E1 -4497.725,E2 -4497.725} C_VEL
LIN {X 0,Y 531.161,Z 339.324,A -85,B 0,C 180,E1 -4500.758,E2 -4500.758} C_VEL
LIN {X 0,Y 531.11,Z 339.33,A -85,B 0,C 180,E1 -4503.034,E2 -4503.034} C_VEL
LIN {X 0,Y 531.088,Z 339.332,A -85,B 0,C 180,E1 -4506.077,E2 -4506.077} C_VEL
LIN {X 0,Y 531.038,Z 339.338,A -85,B 0,C 180,E1 -4509.138,E2 -4509.138} C_VEL
LIN {X 0,Y 531.047,Z 339.339,A -85,B 0,C 180,E1 -4512.225,E2 -4512.225} C_VEL
LIN {X 0,Y 531.003,Z 339.342,A -85,B 0,C 180,E1 -4515.35,E2 -4515.35} C_VEL
LIN {X 0,Y 530.997,Z 339.343,A -85,B 0,C 180,E1 -4518.521,E2 -4518.521} C_VEL
LIN {X 0,Y 531.005,Z 339.342,A -85,B 0,C 180,E1 -4520.938,E2 -4520.938} C_VEL
LIN {X 0,Y 530.987,Z 339.345,A -85,B 0,C 180,E1 -4524.224,E2 -4524.224} C_VEL
LIN {X 0,Y 531.011,Z 339.342,A -85,B 0,C 180,E1 -4526.744,E2 -4526.744} C_VEL
LIN {X 0,Y 530.987,Z 339.346,A -85,B 0,C 180,E1 -4529.323,E2 -4529.323} C_VEL
LIN {X 0,Y 530.977,Z 339.346,A -85,B 0,C 180,E1 -4532.101,E2 -4532.101} C_VEL
LIN {X 0,Y 530.978,Z 339.347,A -85,B 0,C 180,E1 -4534.851,E2 -4534.851} C_VEL
LIN {X 0,Y 530.973,Z 339.347,A -85,B 0,C 180,E1 -4537.508,E2 -4537.508} C_VEL
LIN {X 0,Y 530.992,Z 339.345,A -85,B 0,C 180,E1 -4540.433,E2 -4540.433} C_VEL
LIN {X 0,Y 530.967,Z 339.347,A -85,B 0,C 180,E1 -4543.281,E2 -4543.281} C_VEL
LIN {X 0,Y 530.959,Z 339.349,A -85,B 0,C 180,E1 -4543.565,E2 -4543.565} C_VEL
LIN {X 0,Y 530.29,Z 339.431,A -85,B 0,C 180,E1 -4544.198,E2 -4544.198} C_VEL
LIN {X 0,Y 527.446,Z 339.786,A -85,B 0,C 180,E1 -4545.227,E2 -4545.227} C_VEL
LIN {X 0,Y 525.045,Z 340.087,A -85,B 0,C 180,E1 -4546.056,E2 -4546.056} C_VEL
LIN {X 0,Y 524.012,Z 340.214,A -85,B 0,C 180,E1 -4546.695,E2 -4546.695} C_VEL
LIN {X 0,Y 523.927,Z 340.224,A -85,B 0,C 180,E1 -4546.912,E2 -4546.912} C_VEL
LIN {X 0,Y 523.955,Z 340.22,A -85,B 0,C 180,E1 -4549.92,E2 -4549.92} C_VEL
LIN {X 0,Y 523.911,Z 340.227,A -85,B 0,C 180,E1 -4552.867,E2 -4552.867} C_VEL
LIN {X 0,Y 523.939,Z 340.223,A -85,B 0,C 180,E1 -4555.71,E2 -4555.71} C_VEL
LIN {X 0,Y 523.929,Z 340.225,A -85,B 0,C 180,E1 -4558.456,E2 -4558.456} C_VEL
LIN {X 0,Y 523.942,Z 340.222,A -85,B 0,C 180,E1 -4561.125,E2 -4561.125} C_VEL
LIN {X 0,Y 523.992,Z 340.216,A -85,B 0,C 180,E1 -4563.98,E2 -4563.98} C_VEL
LIN {X 0,Y 523.933,Z 340.225,A -85,B 0,C 180,E1 -4566.27,E2 -4566.27} C_VEL
LIN {X 0,Y 523.953,Z 340.221,A -85,B 0,C 180,E1 -4568.766,E2 -4568.766} C_VEL
LIN {X 0,Y 523.957,Z 340.22,A -85,B 0,C 180,E1 -4571.22,E2 -4571.22} C_VEL
LIN {X 0,Y 523.944,Z 340.222,A -85,B 0,C 180,E1 -4573.639,E2 -4573.639} C_VEL
LIN {X 0,Y 523.946,Z 340.222,A -85,B 0,C 180,E1 -4576.028,E2 -4576.028} C_VEL
LIN {X 0,Y 524.02,Z 340.214,A -85,B 0,C 180,E1 -4578.394,E2 -4578.394} C_VEL
LIN {X 0,Y 524.011,Z 340.214,A -85,B 0,C 180,E1 -4581.516,E2 -4581.516} C_VEL
LIN {X 0,Y 524.103,Z 340.388,A -85,B 0,C 180,E1 -4584.734,E2 -4584.734} C_VEL
LIN {X 0,Y 525.345,Z 345.849,A -85,B 0,C 180,E1 -4584.963,E2 -4584.963} C_VEL
LIN {X 0,Y 525.164,Z 357.813,A -85,B 0,C 180,E1 -4585.49,E2 -4585.49} C_VEL
LIN {X 0,Y 524.923,Z 369.368,A -85,B 0,C 180,E1 -4586.161,E2 -4586.161} C_VEL
LIN {X 0,Y 524.616,Z 380.878,A -85,B 0,C 180,E1 -4587.024,E2 -4587.024} C_VEL
LIN {X 0,Y 524.336,Z 390.166,A -85,B 0,C 180,E1 -4587.887,E2 -4587.887} C_VEL
LIN {X 0,Y 524.061,Z 398.653,A -85,B 0,C 180,E1 -4588.847,E2 -4588.847} C_VEL
LIN {X 0,Y 523.883,Z 406.899,A -85,B 0,C 180,E1 -4589.999,E2 -4589.999} C_VEL
LIN {X 0,Y 523.653,Z 413.543,A -85,B 0,C 180,E1 -4591.153,E2 -4591.153} C_VEL
LIN {X 0,Y 523.502,Z 418.86,A -85,B 0,C 180,E1 -4592.308,E2 -4592.308} C_VEL
LIN {X 0,Y 523.521,Z 423.011,A -85,B 0,C 180,E1 -4593.463,E2 -4593.463} C_VEL
LIN {X 0,Y 523.396,Z 426.162,A -85,B 0,C 180,E1 -4594.621,E2 -4594.621} C_VEL
LIN {X 0,Y 523.43,Z 427.716,A -85,B 0,C 180,E1 -4595.392,E2 -4595.392} C_VEL
LIN {X 0,Y 523.422,Z 429.215,A -85,B 0,C 180,E1 -4596.481,E2 -4596.481} C_VEL
LIN {X 0,Y 523.404,Z 429.979,A -85,B 0,C 180,E1 -4597.716,E2 -4597.716} C_VEL
LIN {X 0,Y 523.347,Z 429.559,A -85,B 0,C 180,E1 -4599.273,E2 -4599.273} C_VEL
LIN {X 0,Y 523.35,Z 428.719,A -85,B 0,C 180,E1 -4600.053,E2 -4600.053} C_VEL
LIN {X 0,Y 523.451,Z 426.226,A -85,B 0,C 180,E1 -4601.441,E2 -4601.441} C_VEL
LIN {X 0,Y 523.484,Z 422.501,A -85,B 0,C 180,E1 -4602.798,E2 -4602.798} C_VEL
LIN {X 0,Y 523.582,Z 418.064,A -85,B 0,C 180,E1 -4603.981,E2 -4603.981} C_VEL
LIN {X 0,Y 523.762,Z 411.365,A -85,B 0,C 180,E1 -4605.347,E2 -4605.347} C_VEL
LIN {X 0,Y 523.92,Z 403.784,A -85,B 0,C 180,E1 -4606.561,E2 -4606.561} C_VEL
LIN {X 0,Y 524.141,Z 396.768,A -85,B 0,C 180,E1 -4607.476,E2 -4607.476} C_VEL
LIN {X 0,Y 524.44,Z 386.638,A -85,B 0,C 180,E1 -4608.558,E2 -4608.558} C_VEL
LIN {X 0,Y 524.745,Z 376.008,A -85,B 0,C 180,E1 -4609.46,E2 -4609.46} C_VEL
LIN {X 0,Y 525.002,Z 364.045,A -85,B 0,C 180,E1 -4610.265,E2 -4610.265} C_VEL
LIN {X 0,Y 525.267,Z 352.233,A -85,B 0,C 180,E1 -4610.868,E2 -4610.868} C_VEL
LIN {X 0,Y 525.184,Z 344.662,A -85,B 0,C 180,E1 -4611.18,E2 -4611.18} C_VEL
LIN {X 0,Y 523.981,Z 340.219,A -85,B 0,C 180,E1 -4611.386,E2 -4611.386} C_VEL
LIN {X 0,Y 523.935,Z 340.225,A -85,B 0,C 180,E1 -4614.571,E2 -4614.571} C_VEL
LIN {X 0,Y 523.95,Z 340.222,A -85,B 0,C 180,E1 -4617.132,E2 -4617.132} C_VEL
LIN {X 0,Y 523.944,Z 340.225,A -85,B 0,C 180,E1 -4619.755,E2 -4619.755} C_VEL
LIN {X 0,Y 523.938,Z 340.227,A -85,B 0,C 180,E1 -4622.449,E2 -4622.449} C_VEL
LIN {X 0,Y 523.922,Z 340.227,A -85,B 0,C 180,E1 -4625.226,E2 -4625.226} C_VEL
LIN {X 0,Y 523.916,Z 340.225,A -85,B 0,C 180,E1 -4628.101,E2 -4628.101} C_VEL
LIN {X 0,Y 523.942,Z 340.223,A -85,B 0,C 180,E1 -4631.091,E2 -4631.091} C_VEL
LIN {X 0,Y 523.942,Z 340.223,A -85,B 0,C 180,E1 -4634.227,E2 -4634.227} C_VEL
LIN {X 0,Y 523.922,Z 340.224,A -85,B 0,C 180,E1 -4636.833,E2 -4636.833} C_VEL
LIN {X 0,Y 523.978,Z 340.217,A -85,B 0,C 180,E1 -4639.923,E2 -4639.923} C_VEL
LIN {X 0,Y 523.911,Z 340.226,A -85,B 0,C 180,E1 -4642.868,E2 -4642.868} C_VEL
LIN {X 0,Y 523.946,Z 340.223,A -85,B 0,C 180,E1 -4645.71,E2 -4645.71} C_VEL
LIN {X 0,Y 523.932,Z 340.219,A -85,B 0,C 180,E1 -4648.456,E2 -4648.456} C_VEL
LIN {X 0,Y 523.95,Z 340.215,A -85,B 0,C 180,E1 -4651.126,E2 -4651.126} C_VEL
LIN {X 0,Y 523.985,Z 340.216,A -85,B 0,C 180,E1 -4653.979,E2 -4653.979} C_VEL
LIN {X 0,Y 523.935,Z 340.223,A -85,B 0,C 180,E1 -4656.27,E2 -4656.27} C_VEL
LIN {X 0,Y 523.946,Z 340.221,A -85,B 0,C 180,E1 -4658.766,E2 -4658.766} C_VEL
LIN {X 0,Y 523.953,Z 340.221,A -85,B 0,C 180,E1 -4661.221,E2 -4661.221} C_VEL
LIN {X 0,Y 523.94,Z 340.222,A -85,B 0,C 180,E1 -4663.639,E2 -4663.639} C_VEL
LIN {X 0,Y 523.945,Z 340.222,A -85,B 0,C 180,E1 -4666.028,E2 -4666.028} C_VEL
LIN {X 0,Y 524.037,Z 340.212,A -85,B 0,C 180,E1 -4668.394,E2 -4668.394} C_VEL
LIN {X 0,Y 524.006,Z 340.215,A -85,B 0,C 180,E1 -4671.516,E2 -4671.516} C_VEL
LIN {X 0,Y 524.083,Z 340.202,A -85,B 0,C 180,E1 -4674.613,E2 -4674.613} C_VEL
LIN {X 0,Y 524.109,Z 340.201,A -85,B 0,C 180,E1 -4677.694,E2 -4677.694} C_VEL
LIN {X 0,Y 524.123,Z 340.198,A -85,B 0,C 180,E1 -4680.768,E2 -4680.768} C_VEL
LIN {X 0,Y 524.072,Z 340.207,A -85,B 0,C 180,E1 -4683.075,E2 -4683.075} C_VEL
LIN {X 0,Y 524.044,Z 340.209,A -85,B 0,C 180,E1 -4686.159,E2 -4686.159} C_VEL
LIN {X 0,Y 523.998,Z 340.215,A -85,B 0,C 180,E1 -4689.262,E2 -4689.262} C_VEL
LIN {X 0,Y 523.999,Z 340.215,A -85,B 0,C 180,E1 -4691.74,E2 -4691.74} C_VEL
LIN {X 0,Y 523.989,Z 340.216,A -85,B 0,C 180,E1 -4695.052,E2 -4695.052} C_VEL
LIN {X 0,Y 523.961,Z 340.219,A -85,B 0,C 180,E1 -4697.969,E2 -4697.969} C_VEL
LIN {X 0,Y 523.969,Z 340.219,A -85,B 0,C 180,E1 -4700.41,E2 -4700.41} C_VEL
LIN {X 0,Y 523.914,Z 340.227,A -85,B 0,C 180,E1 -4702.893,E2 -4702.893} C_VEL
LIN {X 0,Y 523.952,Z 340.223,A -85,B 0,C 180,E1 -4705.419,E2 -4705.419} C_VEL
LIN {X 0,Y 523.968,Z 340.221,A -85,B 0,C 180,E1 -4707.999,E2 -4707.999} C_VEL
LIN {X 0,Y 523.95,Z 340.222,A -85,B 0,C 180,E1 -4710.857,E2 -4710.857} C_VEL
LIN {X 0,Y 523.96,Z 340.22,A -85,B 0,C 180,E1 -4713.736,E2 -4713.736} C_VEL
LIN {X 0,Y 523.923,Z 340.226,A -85,B 0,C 180,E1 -4716.405,E2 -4716.405} C_VEL
LIN {X 0,Y 523.958,Z 340.219,A -85,B 0,C 180,E1 -4719.081,E2 -4719.081} C_VEL
LIN {X 0,Y 523.957,Z 340.219,A -85,B 0,C 180,E1 -4722.119,E2 -4722.119} C_VEL
LIN {X 0,Y 523.955,Z 340.223,A -85,B 0,C 180,E1 -4725.309,E2 -4725.309} C_VEL
LIN {X 0,Y 523.981,Z 340.219,A -85,B 0,C 180,E1 -4728.687,E2 -4728.687} C_VEL
LIN {X 0,Y 523.925,Z 340.228,A -85,B 0,C 180,E1 -4731.655,E2 -4731.655} C_VEL
LIN {X 0,Y 523.922,Z 340.279,A -85,B 0,C 180,E1 -4731.777,E2 -4731.777} C_VEL
LIN {X 0,Y 525.429,Z 348.147,A -85,B 0,C 180,E1 -4733.948,E2 -4733.948} C_VEL
LIN {X 0,Y 525.245,Z 356.567,A -85,B 0,C 180,E1 -4736.056,E2 -4736.056} C_VEL
LIN {X 0,Y 524.867,Z 370.592,A -85,B 0,C 180,E1 -4739.415,E2 -4739.415} C_VEL
LIN {X 0,Y 524.628,Z 384.164,A -85,B 0,C 180,E1 -4742.525,E2 -4742.525} C_VEL
LIN {X 0,Y 524.399,Z 398.467,A -85,B 0,C 180,E1 -4745.691,E2 -4745.691} C_VEL
LIN {X 0,Y 524.223,Z 412.728,A -85,B 0,C 180,E1 -4748.779,E2 -4748.779} C_VEL
LIN {X 0,Y 524.049,Z 426.178,A -85,B 0,C 180,E1 -4751.63,E2 -4751.63} C_VEL
LIN {X 0,Y 523.886,Z 439.693,A -85,B 0,C 180,E1 -4754.437,E2 -4754.437} C_VEL
LIN {X 0,Y 523.793,Z 448.398,A -85,B 0,C 180,E1 -4756.247,E2 -4756.247} C_VEL
LIN {X 0,Y 525.391,Z 460.254,A -85,B 0,C 180,E1 -4756.536,E2 -4756.536} C_VEL
LIN {X 0,Y 525.189,Z 473.389,A -85,B 0,C 180,E1 -4756.95,E2 -4756.95} C_VEL
LIN {X 0,Y 524.954,Z 484.513,A -85,B 0,C 180,E1 -4757.435,E2 -4757.435} C_VEL
LIN {X 0,Y 524.67,Z 496.725,A -85,B 0,C 180,E1 -4758.131,E2 -4758.131} C_VEL
LIN {X 0,Y 524.392,Z 508.447,A -85,B 0,C 180,E1 -4758.991,E2 -4758.991} C_VEL
LIN {X 0,Y 524.074,Z 519.076,A -85,B 0,C 180,E1 -4759.961,E2 -4759.961} C_VEL
LIN {X 0,Y 523.873,Z 527.703,A -85,B 0,C 180,E1 -4760.931,E2 -4760.931} C_VEL
LIN {X 0,Y 523.687,Z 536.125,A -85,B 0,C 180,E1 -4762.094,E2 -4762.094} C_VEL
LIN {X 0,Y 523.574,Z 541.842,A -85,B 0,C 180,E1 -4763.062,E2 -4763.062} C_VEL
LIN {X 0,Y 523.544,Z 547.368,A -85,B 0,C 180,E1 -4764.222,E2 -4764.222} C_VEL
LIN {X 0,Y 523.36,Z 551.678,A -85,B 0,C 180,E1 -4765.379,E2 -4765.379} C_VEL
LIN {X 0,Y 523.443,Z 553.959,A -85,B 0,C 180,E1 -4766.151,E2 -4766.151} C_VEL
LIN {X 0,Y 523.367,Z 555.808,A -85,B 0,C 180,E1 -4766.922,E2 -4766.922} C_VEL
LIN {X 0,Y 523.335,Z 557.193,A -85,B 0,C 180,E1 -4767.692,E2 -4767.692} C_VEL
LIN {X 0,Y 523.25,Z 558.785,A -85,B 0,C 180,E1 -4769.231,E2 -4769.231} C_VEL
LIN {X 0,Y 523.246,Z 559,A -85,B 0,C 180,E1 -4770.001,E2 -4770.001} C_VEL
LIN {X 0,Y 523.275,Z 558.182,A -85,B 0,C 180,E1 -4771.54,E2 -4771.54} C_VEL
LIN {X 0,Y 523.335,Z 557.195,A -85,B 0,C 180,E1 -4772.309,E2 -4772.309} C_VEL
LIN {X 0,Y 523.367,Z 555.809,A -85,B 0,C 180,E1 -4773.08,E2 -4773.08} C_VEL
LIN {X 0,Y 523.441,Z 552.893,A -85,B 0,C 180,E1 -4774.235,E2 -4774.235} C_VEL
LIN {X 0,Y 523.464,Z 548.946,A -85,B 0,C 180,E1 -4775.393,E2 -4775.393} C_VEL
LIN {X 0,Y 523.523,Z 543.711,A -85,B 0,C 180,E1 -4776.581,E2 -4776.581} C_VEL
LIN {X 0,Y 523.665,Z 537.371,A -85,B 0,C 180,E1 -4777.713,E2 -4777.713} C_VEL
LIN {X 0,Y 523.846,Z 529.213,A -85,B 0,C 180,E1 -4778.876,E2 -4778.876} C_VEL
LIN {X 0,Y 524.034,Z 520.902,A -85,B 0,C 180,E1 -4779.846,E2 -4779.846} C_VEL
LIN {X 0,Y 524.341,Z 510.793,A -85,B 0,C 180,E1 -4780.816,E2 -4780.816} C_VEL
LIN {X 0,Y 524.621,Z 499.4,A -85,B 0,C 180,E1 -4781.69,E2 -4781.69} C_VEL
LIN {X 0,Y 524.875,Z 488.241,A -85,B 0,C 180,E1 -4782.371,E2 -4782.371} C_VEL
LIN {X 0,Y 525.13,Z 475.911,A -85,B 0,C 180,E1 -4782.955,E2 -4782.955} C_VEL
LIN {X 0,Y 525.364,Z 462.995,A -85,B 0,C 180,E1 -4783.392,E2 -4783.392} C_VEL
LIN {X 0,Y 525.091,Z 457.67,A -85,B 0,C 180,E1 -4783.534,E2 -4783.534} C_VEL
LIN {X 0,Y 523.796,Z 448.435,A -85,B 0,C 180,E1 -4783.754,E2 -4783.754} C_VEL
LIN {X 0,Y 523.986,Z 434.041,A -85,B 0,C 180,E1 -4786.761,E2 -4786.761} C_VEL
LIN {X 0,Y 524.148,Z 419.093,A -85,B 0,C 180,E1 -4789.886,E2 -4789.886} C_VEL
LIN {X 0,Y 524.337,Z 405.209,A -85,B 0,C 180,E1 -4792.874,E2 -4792.874} C_VEL
LIN {X 0,Y 524.513,Z 392.025,A -85,B 0,C 180,E1 -4795.766,E2 -4795.766} C_VEL
LIN {X 0,Y 524.742,Z 378.402,A -85,B 0,C 180,E1 -4798.827,E2 -4798.827} C_VEL
LIN {X 0,Y 524.996,Z 364.965,A -85,B 0,C 180,E1 -4801.924,E2 -4801.924} C_VEL
LIN {X 0,Y 525.402,Z 350.728,A -85,B 0,C 180,E1 -4805.317,E2 -4805.317} C_VEL
LIN {X 0,Y 524.994,Z 345.788,A -85,B 0,C 180,E1 -4806.562,E2 -4806.562} C_VEL
LIN {X 0,Y 523.928,Z 340.224,A -85,B 0,C 180,E1 -4808.044,E2 -4808.044} C_VEL
LIN {X 0,Y 523.946,Z 340.222,A -85,B 0,C 180,E1 -4811.092,E2 -4811.092} C_VEL
LIN {X 0,Y 523.947,Z 340.223,A -85,B 0,C 180,E1 -4814.228,E2 -4814.228} C_VEL
LIN {X 0,Y 523.922,Z 340.225,A -85,B 0,C 180,E1 -4816.833,E2 -4816.833} C_VEL
LIN {X 0,Y 523.947,Z 340.222,A -85,B 0,C 180,E1 -4818.908,E2 -4818.908} C_VEL
LIN {X 0,Y 523.922,Z 340.225,A -85,B 0,C 180,E1 -4821.899,E2 -4821.899} C_VEL
LIN {X 0,Y 523.93,Z 340.225,A -85,B 0,C 180,E1 -4824.911,E2 -4824.911} C_VEL
LIN {X 0,Y 523.948,Z 340.22,A -85,B 0,C 180,E1 -4827.679,E2 -4827.679} C_VEL
LIN {X 0,Y 523.96,Z 340.222,A -85,B 0,C 180,E1 -4830.677,E2 -4830.677} C_VEL
LIN {X 0,Y 523.979,Z 340.217,A -85,B 0,C 180,E1 -4833.729,E2 -4833.729} C_VEL
LIN {X 0,Y 523.943,Z 340.223,A -85,B 0,C 180,E1 -4836.271,E2 -4836.271} C_VEL
LIN {X 0,Y 523.951,Z 340.222,A -85,B 0,C 180,E1 -4838.767,E2 -4838.767} C_VEL
LIN {X 0,Y 523.953,Z 340.22,A -85,B 0,C 180,E1 -4841.221,E2 -4841.221} C_VEL
LIN {X 0,Y 523.939,Z 340.221,A -85,B 0,C 180,E1 -4843.639,E2 -4843.639} C_VEL
LIN {X 0,Y 523.946,Z 340.221,A -85,B 0,C 180,E1 -4846.028,E2 -4846.028} C_VEL
LIN {X 0,Y 524.019,Z 340.213,A -85,B 0,C 180,E1 -4848.394,E2 -4848.394} C_VEL
LIN {X 0,Y 524.008,Z 340.212,A -85,B 0,C 180,E1 -4851.516,E2 -4851.516} C_VEL
LIN {X 0,Y 524.089,Z 340.204,A -85,B 0,C 180,E1 -4854.614,E2 -4854.614} C_VEL
LIN {X 0,Y 524.114,Z 340.202,A -85,B 0,C 180,E1 -4857.695,E2 -4857.695} C_VEL
LIN {X 0,Y 524.131,Z 340.2,A -85,B 0,C 180,E1 -4860.768,E2 -4860.768} C_VEL
LIN {X 0,Y 524.077,Z 340.206,A -85,B 0,C 180,E1 -4863.075,E2 -4863.075} C_VEL
LIN {X 0,Y 524.051,Z 340.209,A -85,B 0,C 180,E1 -4866.159,E2 -4866.159} C_VEL
LIN {X 0,Y 524.006,Z 340.214,A -85,B 0,C 180,E1 -4869.262,E2 -4869.262} C_VEL
LIN {X 0,Y 524.009,Z 340.214,A -85,B 0,C 180,E1 -4871.739,E2 -4871.739} C_VEL
LIN {X 0,Y 524,Z 340.213,A -85,B 0,C 180,E1 -4875.052,E2 -4875.052} C_VEL
LIN {X 0,Y 523.971,Z 340.22,A -85,B 0,C 180,E1 -4877.969,E2 -4877.969} C_VEL
LIN {X 0,Y 523.978,Z 340.217,A -85,B 0,C 180,E1 -4880.41,E2 -4880.41} C_VEL
LIN {X 0,Y 523.922,Z 340.223,A -85,B 0,C 180,E1 -4882.893,E2 -4882.893} C_VEL
LIN {X 0,Y 523.96,Z 340.22,A -85,B 0,C 180,E1 -4885.419,E2 -4885.419} C_VEL
LIN {X 0,Y 523.966,Z 340.22,A -85,B 0,C 180,E1 -4887.999,E2 -4887.999} C_VEL
LIN {X 0,Y 523.951,Z 340.22,A -85,B 0,C 180,E1 -4890.855,E2 -4890.855} C_VEL
LIN {X 0,Y 523.966,Z 340.22,A -85,B 0,C 180,E1 -4893.735,E2 -4893.735} C_VEL
LIN {X 0,Y 523.91,Z 340.225,A -85,B 0,C 180,E1 -4896.401,E2 -4896.401} C_VEL
LIN {X 0,Y 523.931,Z 340.225,A -85,B 0,C 180,E1 -4899.084,E2 -4899.084} C_VEL
LIN {X 0,Y 523.96,Z 340.22,A -85,B 0,C 180,E1 -4902.119,E2 -4902.119} C_VEL
LIN {X 0,Y 523.962,Z 340.22,A -85,B 0,C 180,E1 -4905.309,E2 -4905.309} C_VEL
LIN {X 0,Y 523.927,Z 340.224,A -85,B 0,C 180,E1 -4906.912,E2 -4906.912} C_VEL
LIN {X 0,Y 523.26,Z 340.308,A -85,B 0,C 180,E1 -4907.553,E2 -4907.553} C_VEL
LIN {X 0,Y 520.418,Z 340.661,A -85,B 0,C 180,E1 -4908.595,E2 -4908.595} C_VEL
LIN {X 0,Y 518.013,Z 340.963,A -85,B 0,C 180,E1 -4909.434,E2 -4909.434} C_VEL
LIN {X 0,Y 516.975,Z 341.091,A -85,B 0,C 180,E1 -4910.082,E2 -4910.082} C_VEL
LIN {X 0,Y 516.888,Z 341.101,A -85,B 0,C 180,E1 -4910.301,E2 -4910.301} C_VEL
LIN {X 0,Y 516.86,Z 341.105,A -85,B 0,C 180,E1 -4913.346,E2 -4913.346} C_VEL
LIN {X 0,Y 516.914,Z 341.098,A -85,B 0,C 180,E1 -4916.121,E2 -4916.121} C_VEL
LIN {X 0,Y 516.897,Z 341.1,A -85,B 0,C 180,E1 -4918.936,E2 -4918.936} C_VEL
LIN {X 0,Y 516.922,Z 341.097,A -85,B 0,C 180,E1 -4921.584,E2 -4921.584} C_VEL
LIN {X 0,Y 516.939,Z 341.094,A -85,B 0,C 180,E1 -4924.211,E2 -4924.211} C_VEL
LIN {X 0,Y 516.873,Z 341.103,A -85,B 0,C 180,E1 -4926.776,E2 -4926.776} C_VEL
LIN {X 0,Y 516.947,Z 341.093,A -85,B 0,C 180,E1 -4929.731,E2 -4929.731} C_VEL
LIN {X 0,Y 516.929,Z 341.097,A -85,B 0,C 180,E1 -4932.596,E2 -4932.596} C_VEL
LIN {X 0,Y 516.95,Z 341.095,A -85,B 0,C 180,E1 -4935.03,E2 -4935.03} C_VEL
LIN {X 0,Y 516.973,Z 341.09,A -85,B 0,C 180,E1 -4938.233,E2 -4938.233} C_VEL
LIN {X 0,Y 516.976,Z 341.09,A -85,B 0,C 180,E1 -4941.399,E2 -4941.399} C_VEL
LIN {X 0,Y 517.029,Z 341.084,A -85,B 0,C 180,E1 -4944.539,E2 -4944.539} C_VEL
LIN {X 0,Y 518.478,Z 347.015,A -85,B 0,C 180,E1 -4944.798,E2 -4944.798} C_VEL
LIN {X 0,Y 518.295,Z 358.901,A -85,B 0,C 180,E1 -4945.333,E2 -4945.333} C_VEL
LIN {X 0,Y 518.035,Z 370.394,A -85,B 0,C 180,E1 -4946.013,E2 -4946.013} C_VEL
LIN {X 0,Y 517.697,Z 381.876,A -85,B 0,C 180,E1 -4946.887,E2 -4946.887} C_VEL
LIN {X 0,Y 517.368,Z 392.091,A -85,B 0,C 180,E1 -4947.859,E2 -4947.859} C_VEL
LIN {X 0,Y 517.119,Z 400.368,A -85,B 0,C 180,E1 -4948.831,E2 -4948.831} C_VEL
LIN {X 0,Y 516.895,Z 408.43,A -85,B 0,C 180,E1 -4949.999,E2 -4949.999} C_VEL
LIN {X 0,Y 516.642,Z 414.955,A -85,B 0,C 180,E1 -4951.169,E2 -4951.169} C_VEL
LIN {X 0,Y 516.501,Z 420.161,A -85,B 0,C 180,E1 -4952.339,E2 -4952.339} C_VEL
LIN {X 0,Y 516.491,Z 424.216,A -85,B 0,C 180,E1 -4953.51,E2 -4953.51} C_VEL
LIN {X 0,Y 516.371,Z 427.271,A -85,B 0,C 180,E1 -4954.684,E2 -4954.684} C_VEL
LIN {X 0,Y 516.411,Z 428.781,A -85,B 0,C 180,E1 -4955.466,E2 -4955.466} C_VEL
LIN {X 0,Y 516.377,Z 430.134,A -85,B 0,C 180,E1 -4956.509,E2 -4956.509} C_VEL
LIN {X 0,Y 516.362,Z 430.871,A -85,B 0,C 180,E1 -4957.822,E2 -4957.822} C_VEL
LIN {X 0,Y 516.344,Z 430.809,A -85,B 0,C 180,E1 -4958.61,E2 -4958.61} C_VEL
LIN {X 0,Y 516.309,Z 430.33,A -85,B 0,C 180,E1 -4959.4,E2 -4959.4} C_VEL
LIN {X 0,Y 516.403,Z 428.145,A -85,B 0,C 180,E1 -4960.983,E2 -4960.983} C_VEL
LIN {X 0,Y 516.448,Z 425.402,A -85,B 0,C 180,E1 -4962.176,E2 -4962.176} C_VEL
LIN {X 0,Y 516.498,Z 421.616,A -85,B 0,C 180,E1 -4963.374,E2 -4963.374} C_VEL
LIN {X 0,Y 516.66,Z 416.662,A -85,B 0,C 180,E1 -4964.575,E2 -4964.575} C_VEL
LIN {X 0,Y 516.821,Z 410.377,A -85,B 0,C 180,E1 -4965.781,E2 -4965.781} C_VEL
LIN {X 0,Y 517.048,Z 402.41,A -85,B 0,C 180,E1 -4966.991,E2 -4966.991} C_VEL
